KUKA KRL program: MyProgram_216().src

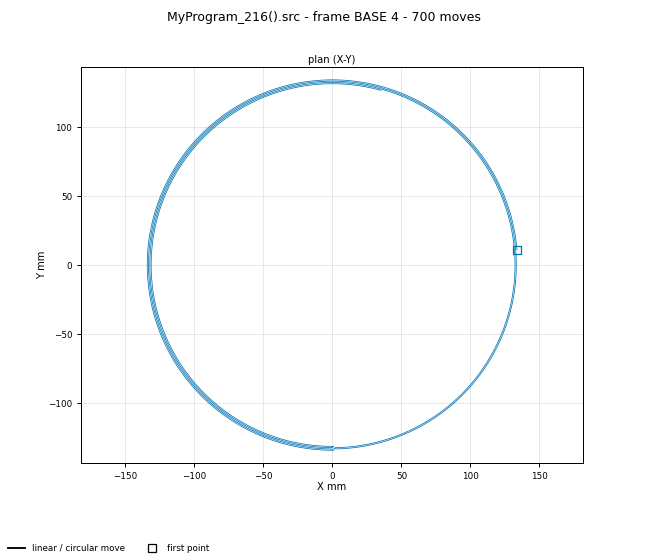
[picture p0: tool path of MyProgram_216().src in frame BASE 4, 700 of 700 moves have a stored position in this frame; points joined in program order, loops and branches not executed]
&ACCESS RVP
&REL 1
&PARAM TEMPLATE = C:\KRC\Roboter\Template\vorgabe
&PARAM EDITMASK = *
DEF MyProgram_216()
; ---- Setting reference (Base) ----
$BASE = BASE_DATA[4]

; --------------------------
; ---- Setting tool (TCP) ----
$TOOL = TOOL_DATA[3]
; --------------------------

$VEL.CP = VEL_APROX_PRINT
Startdeposition()
$VEL.CP = VEL_PRINT
LIN {X 133.7313,Y 11.0873,Z 152,A 1.5127,B 24.9579,C -1.4999,E1 25.1592,E2 444.9468} C_DIS
LIN {X 133.4155,Y 14.396,Z 152,A 2.9886,B 24.9574,C -1.5078,E1 25.1587,E2 443.4612} C_DIS
LIN {X 132.9448,Y 18.2524,Z 152,A 4.7216,B 24.9569,C -1.5174,E1 25.1581,E2 441.7159} C_DIS
LIN {X 132.4358,Y 21.6308,Z 152,A 6.0104,B 24.9571,C -1.5126,E1 25.1576,E2 440.446} C_DIS
LIN {X 131.8421,Y 24.9924,Z 152,A 7.5184,B 24.9567,C -1.5201,E1 25.1568,E2 438.9291} C_DIS
LIN {X 131.1946,Y 28.1941,Z 152,A 8.8428,B 24.9567,C -1.5206,E1 25.156,E2 437.6112} C_DIS
LIN {X 130.4813,Y 31.3296,Z 152,A 10.2545,B 24.9563,C -1.5272,E1 25.1551,E2 436.1923} C_DIS
LIN {X 129.7343,Y 34.2927,Z 152,A 11.61,B 24.9559,C -1.5341,E1 25.1542,E2 434.8282} C_DIS
LIN {X 128.7032,Y 37.9795,Z 152,A 13.1947,B 24.9558,C -1.5364,E1 25.153,E2 433.2471} C_DIS
LIN {X 127.4835,Y 41.8939,Z 152,A 14.9747,B 24.9554,C -1.5435,E1 25.1514,E2 431.4606} C_DIS
LIN {X 126.3534,Y 45.1861,Z 152,A 16.3661,B 24.9554,C -1.5427,E1 25.1502,E2 430.0789} C_DIS
LIN {X 125.2613,Y 48.1324,Z 152,A 17.8112,B 24.9548,C -1.5525,E1 25.1487,E2 428.6186} C_DIS
LIN {X 123.987,Y 51.3249,Z 152,A 19.2654,B 24.9546,C -1.5562,E1 25.1472,E2 427.1639} C_DIS
LIN {X 122.6392,Y 54.4665,Z 152,A 20.5859,B 24.9548,C -1.5527,E1 25.1457,E2 425.8588} C_DIS
LIN {X 121.2451,Y 57.5031,Z 152,A 22.076,B 24.9544,C -1.5604,E1 25.1439,E2 424.3586} C_DIS
LIN {X 119.8144,Y 60.4284,Z 152,A 23.4608,B 24.9542,C -1.5641,E1 25.1422,E2 422.9724} C_DIS
LIN {X 118.1627,Y 63.5998,Z 152,A 24.9583,B 24.954,C -1.5667,E1 25.1403,E2 421.4766} C_DIS
LIN {X 116.2257,Y 67.0745,Z 152,A 26.7209,B 24.9535,C -1.575,E1 25.1378,E2 419.7036} C_DIS
LIN {X 114.0335,Y 70.7371,Z 152,A 28.4898,B 24.9535,C -1.577,E1 25.1352,E2 417.9391} C_DIS
LIN {X 111.8163,Y 74.193,Z 152,A 30.2878,B 24.953,C -1.5841,E1 25.1325,E2 416.1331} C_DIS
LIN {X 109.4013,Y 77.7103,Z 152,A 32.1022,B 24.9527,C -1.5885,E1 25.1296,E2 414.3175} C_DIS
LIN {X 106.8036,Y 81.2433,Z 152,A 33.9859,B 24.9524,C -1.5938,E1 25.1264,E2 412.4301} C_DIS
LIN {X 104.2349,Y 84.5136,Z 152,A 35.6507,B 24.9525,C -1.592,E1 25.1235,E2 410.7773} C_DIS
LIN {X 101.537,Y 87.7362,Z 152,A 37.4625,B 24.9522,C -1.5973,E1 25.1203,E2 408.9614} C_DIS
LIN {X 98.7559,Y 90.855,Z 152,A 39.2295,B 24.952,C -1.6005,E1 25.117,E2 407.1947} C_DIS
LIN {X 95.9879,Y 93.775,Z 152,A 40.9822,B 24.9517,C -1.6063,E1 25.1135,E2 405.4359} C_DIS
LIN {X 93.1738,Y 96.5714,Z 152,A 42.6108,B 24.9517,C -1.6063,E1 25.1103,E2 403.8139} C_DIS
LIN {X 90.3468,Y 99.2213,Z 152,A 44.2646,B 24.9514,C -1.6098,E1 25.1069,E2 402.1588} C_DIS
LIN {X 87.5654,Y 101.6841,Z 152,A 45.9253,B 24.951,C -1.6171,E1 25.1034,E2 400.4874} C_DIS
LIN {X 83.9511,Y 104.6886,Z 152,A 47.8636,B 24.951,C -1.6171,E1 25.0992,E2 398.5561} C_DIS
LIN {X 80.9004,Y 107.063,Z 152,A 49.53,B 24.9508,C -1.6211,E1 25.0955,E2 396.8865} C_DIS
LIN {X 77.4008,Y 109.6196,Z 152,A 51.379,B 24.9506,C -1.6243,E1 25.0913,E2 395.0364} C_DIS
LIN {X 73.8298,Y 112.0559,Z 152,A 53.2038,B 24.9504,C -1.6263,E1 25.0871,E2 393.2132} C_DIS
LIN {X 70.4565,Y 114.2075,Z 152,A 54.9256,B 24.9502,C -1.6297,E1 25.083,E2 391.4888} C_DIS
LIN {X 67.0207,Y 116.2568,Z 152,A 56.6299,B 24.9501,C -1.6321,E1 25.0789,E2 389.7841} C_DIS
LIN {X 63.2307,Y 118.361,Z 152,A 58.4829,B 24.9499,C -1.6348,E1 25.0744,E2 387.93} C_DIS
LIN {X 59.7834,Y 120.1374,Z 152,A 60.1274,B 24.9499,C -1.6364,E1 25.0703,E2 386.2863} C_DIS
LIN {X 56.5816,Y 121.6776,Z 152,A 61.5102,B 24.9502,C -1.631,E1 25.0668,E2 384.9197} C_DIS
LIN {X 53.2944,Y 123.1525,Z 152,A 63.0006,B 24.9502,C -1.6302,E1 25.063,E2 383.4348} C_DIS
LIN {X 50.1244,Y 124.4765,Z 152,A 64.5712,B 24.9498,C -1.6373,E1 25.0589,E2 381.851} C_DIS
LIN {X 46.3326,Y 125.9395,Z 152,A 66.2773,B 24.9498,C -1.6374,E1 25.0545,E2 380.1483} C_DIS
LIN {X 43.1022,Y 127.0811,Z 152,A 67.8485,B 24.9493,C -1.6445,E1 25.0503,E2 378.5634} C_DIS
LIN {X 39.4563,Y 128.258,Z 152,A 69.3935,B 24.9495,C -1.6411,E1 25.0462,E2 377.0294} C_DIS
LIN {X 35.9558,Y 129.283,Z 152,A 70.9825,B 24.9494,C -1.6439,E1 25.0419,E2 375.4365} C_DIS
LIN {X 31.7004,Y 130.3919,Z 152,A 72.7739,B 24.9496,C -1.6404,E1 25.0371,E2 373.6559} C_DIS
LIN {X 28.3792,Y 131.1546,Z 152,A 74.2645,B 24.9494,C -1.6431,E1 25.033,E2 372.161} C_DIS
LIN {X 24.8262,Y 131.8739,Z 152,A 75.9447,B 24.9489,C -1.6508,E1 25.0284,E2 370.4646} C_DIS
LIN {X 20.913,Y 132.5508,Z 152,A 77.5552,B 24.9492,C -1.6468,E1 25.024,E2 368.865} C_DIS
LIN {X 17.2525,Y 133.0764,Z 152,A 79.1159,B 24.9492,C -1.6463,E1 25.0197,E2 367.307} C_DIS
LIN {X 12.8731,Y 133.5711,Z 152,A 80.9369,B 24.9494,C -1.6434,E1 25.0146,E2 365.4941} C_DIS
LIN {X 9.2958,Y 133.8685,Z 152,A 82.5431,B 24.9492,C -1.6473,E1 25.0101,E2 363.8794} C_DIS
LIN {X 5.4111,Y 134.081,Z 152,A 84.1584,B 24.9493,C -1.6448,E1 25.0056,E2 362.2704} C_DIS
LIN {X 1.5384,Y 134.1831,Z 152,A 85.898,B 24.949,C -1.6491,E1 25.0008,E2 360.5211} C_DIS
LIN {X -2.3618,Y 134.1694,Z 152,A 87.5071,B 24.9492,C -1.6458,E1 24.9963,E2 358.9198} C_DIS
LIN {X -6.3709,Y 134.0392,Z 152,A 89.2472,B 24.9492,C -1.6466,E1 24.9914,E2 357.1773} C_DIS
LIN {X -10.1962,Y 133.8028,Z 152,A 90.829,B 24.9494,C -1.6431,E1 24.987,E2 355.6033} C_DIS
LIN {X -14.1568,Y 133.4413,Z 152,A 92.4422,B 24.9497,C -1.6378,E1 24.9826,E2 354.0017} C_DIS
LIN {X -16.9888,Y 133.1109,Z 152,A 93.8388,B 24.9492,C -1.6464,E1 24.9787,E2 352.5839} C_DIS
LIN {X -20.9159,Y 132.5504,Z 152,A 95.4997,B 24.9494,C -1.6435,E1 24.9741,E2 350.9283} C_DIS
LIN {X -24.8462,Y 131.87,Z 152,A 97.0933,B 24.9498,C -1.6365,E1 24.9698,E2 349.3497} C_DIS
LIN {X -28.2027,Y 131.1927,Z 152,A 98.6253,B 24.9497,C -1.6389,E1 24.9655,E2 347.8102} C_DIS
LIN {X -31.5524,Y 130.4276,Z 152,A 100.1386,B 24.9497,C -1.6399,E1 24.9614,E2 346.2926} C_DIS
LIN {X -35.7751,Y 129.3336,Z 152,A 102.0205,B 24.9497,C -1.6389,E1 24.9563,E2 344.4101} C_DIS
LIN {X -39.2856,Y 128.3102,Z 152,A 103.4854,B 24.9501,C -1.6322,E1 24.9525,E2 342.9587} C_DIS
LIN {X -42.0322,Y 127.4375,Z 152,A 104.8372,B 24.9498,C -1.6369,E1 24.9488,E2 341.5932} C_DIS
LIN {X -45.8569,Y 126.1116,Z 152,A 106.5663,B 24.9499,C -1.6347,E1 24.9443,E2 339.8659} C_DIS
LIN {X -49.5966,Y 124.6892,Z 152,A 108.286,B 24.95,C -1.6329,E1 24.9398,E2 338.1469} C_DIS
LIN {X -53.1698,Y 123.2064,Z 152,A 109.8139,B 24.9506,C -1.6242,E1 24.9359,E2 336.6361} C_DIS
LIN {X -56.2408,Y 121.8352,Z 152,A 111.2411,B 24.9507,C -1.6215,E1 24.9323,E2 335.2117} C_DIS
LIN {X -59.2294,Y 120.4107,Z 152,A 112.6995,B 24.9507,C -1.6215,E1 24.9286,E2 333.7495} C_DIS
LIN {X -62.2741,Y 118.8645,Z 152,A 114.1552,B 24.9509,C -1.6189,E1 24.925,E2 332.2961} C_DIS
LIN {X -65.655,Y 117.0333,Z 152,A 115.9269,B 24.9507,C -1.6226,E1 24.9207,E2 330.5107} C_DIS
LIN {X -69.6111,Y 114.7244,Z 152,A 117.8168,B 24.9511,C -1.6156,E1 24.9162,E2 328.6315} C_DIS
LIN {X -72.8488,Y 112.6964,Z 152,A 119.5085,B 24.9511,C -1.6155,E1 24.9122,E2 326.9348} C_DIS
LIN {X -76.4014,Y 110.3189,Z 152,A 121.2229,B 24.9517,C -1.6062,E1 24.9082,E2 325.2366} C_DIS
LIN {X -80.5,Y 107.3651,Z 152,A 123.7555,B 24.9508,C -1.6205,E1 24.9024,E2 322.661} C_DIS
LIN {X -83.2101,Y 105.2786,Z 152,A 124.9589,B 24.9518,C -1.6044,E1 24.8999,E2 321.4916} C_DIS
LIN {X -86.56,Y 102.542,Z 152,A 126.6153,B 24.9526,C -1.5907,E1 24.8964,E2 319.8614} C_DIS
LIN {X -89.6519,Y 99.8494,Z 152,A 128.5412,B 24.9523,C -1.5954,E1 24.8923,E2 317.9169} C_DIS
LIN {X -92.4999,Y 97.2173,Z 152,A 130.213,B 24.9525,C -1.5922,E1 24.8889,E2 316.2458} C_DIS
LIN {X -95.3781,Y 94.3951,Z 152,A 131.9585,B 24.9527,C -1.5891,E1 24.8854,E2 314.5001} C_DIS
LIN {X -99.147,Y 90.4287,Z 152,A 134.3393,B 24.9529,C -1.5854,E1 24.8809,E2 312.1178} C_DIS
LIN {X -101.8173,Y 87.4107,Z 152,A 136.0686,B 24.9531,C -1.5813,E1 24.8777,E2 310.3904} C_DIS
LIN {X -104.5409,Y 84.1343,Z 152,A 137.8461,B 24.9536,C -1.5744,E1 24.8746,E2 308.6213} C_DIS
LIN {X -107.0195,Y 80.958,Z 152,A 139.593,B 24.9538,C -1.571,E1 24.8716,E2 306.874} C_DIS
LIN {X -109.3032,Y 77.8474,Z 152,A 141.2807,B 24.9539,C -1.5683,E1 24.8689,E2 305.1844} C_DIS
LIN {X -111.7611,Y 74.2757,Z 152,A 143.0987,B 24.9543,C -1.5614,E1 24.866,E2 303.3739} C_DIS
LIN {X -113.9277,Y 70.9071,Z 152,A 144.8218,B 24.9546,C -1.5571,E1 24.8635,E2 301.6523} C_DIS
LIN {X -115.9039,Y 67.6298,Z 152,A 146.5135,B 24.9546,C -1.5551,E1 24.861,E2 299.9566} C_DIS
LIN {X -117.7597,Y 64.3429,Z 152,A 148.0857,B 24.9551,C -1.5484,E1 24.8589,E2 298.3922} C_DIS
LIN {X -119.5065,Y 61.0332,Z 152,A 149.6708,B 24.9554,C -1.5429,E1 24.8569,E2 296.8116} C_DIS
LIN {X -121.0233,Y 57.9674,Z 152,A 151.1342,B 24.9556,C -1.5386,E1 24.8551,E2 295.3505} C_DIS
LIN {X -122.4213,Y 54.9536,Z 152,A 152.4985,B 24.9561,C -1.5316,E1 24.8535,E2 293.9956} C_DIS
LIN {X -123.7101,Y 51.9879,Z 152,A 153.9859,B 24.956,C -1.5325,E1 24.8519,E2 292.4977} C_DIS
LIN {X -124.9732,Y 48.8736,Z 152,A 155.4287,B 24.9562,C -1.5284,E1 24.8504,E2 291.0567} C_DIS
LIN {X -126.2429,Y 45.4928,Z 152,A 156.9066,B 24.9567,C -1.5203,E1 24.849,E2 289.5896} C_DIS
LIN {X -127.1836,Y 42.7946,Z 152,A 158.2602,B 24.9565,C -1.523,E1 24.8478,E2 288.222} C_DIS
LIN {X -128.3048,Y 39.3032,Z 152,A 159.6429,B 24.9573,C -1.509,E1 24.8466,E2 286.8647} C_DIS
LIN {X -129.2501,Y 36.0735,Z 152,A 161.2232,B 24.9573,C -1.5114,E1 24.8454,E2 285.2695} C_DIS
LIN {X -130.2973,Y 32.0928,Z 152,A 162.9399,B 24.9576,C -1.5036,E1 24.8442,E2 283.5613} C_DIS
LIN {X -131.1463,Y 28.4176,Z 152,A 164.5492,B 24.9579,C -1.4983,E1 24.8432,E2 281.9552} C_DIS
LIN {X -131.7346,Y 25.5545,Z 152,A 165.8929,B 24.9579,C -1.4989,E1 24.8425,E2 280.6022} C_DIS
LIN {X -132.3897,Y 21.9072,Z 152,A 167.4388,B 24.9583,C -1.4919,E1 24.8418,E2 279.0637} C_DIS
LIN {X -132.9993,Y 17.8409,Z 152,A 169.204,B 24.9586,C -1.4866,E1 24.8411,E2 277.3007} C_DIS
LIN {X -133.4252,Y 14.306,Z 152,A 170.7541,B 24.9588,C -1.483,E1 24.8406,E2 275.7498} C_DIS
LIN {X -133.79,Y 10.371,Z 152,A 172.5007,B 24.9589,C -1.4804,E1 24.8402,E2 273.9991} C_DIS
LIN {X -134.0268,Y 6.618,Z 152,A 174.0782,B 24.9593,C -1.4737,E1 24.8399,E2 272.428} C_DIS
LIN {X -134.1689,Y 2.3895,Z 152,A 175.8019,B 24.9599,C -1.4636,E1 24.8399,E2 270.7179} C_DIS
LIN {X -134.1918,Y -0.3012,Z 152,A 177.13,B 24.9596,C -1.4686,E1 24.8398,E2 269.3699} C_DIS
LIN {X -134.1223,Y -4.3022,Z 152,A 178.8913,B 24.9598,C -1.4656,E1 24.8399,E2 267.6052} C_DIS
LIN {X -133.9167,Y -8.5657,Z 152,A -179.4068,B 24.9604,C -1.4537,E1 24.8402,E2 265.9215} C_DIS
LIN {X -133.5825,Y -12.7544,Z 152,A -177.6549,B 24.9608,C -1.4457,E1 24.8406,E2 264.178} C_DIS
LIN {X -133.2718,Y -15.6723,Z 152,A -176.3213,B 24.9608,C -1.4456,E1 24.841,E2 262.8367} C_DIS
LIN {X -132.8013,Y -19.2565,Z 152,A -174.7809,B 24.9611,C -1.4404,E1 24.8416,E2 261.2994} C_DIS
LIN {X -132.3608,Y -22.0803,Z 152,A -172.8087,B 24.9593,C -1.4738,E1 24.8426,E2 259.2359} C_DIS
LIN {X -131.2989,Y -27.7109,Z 152,A -171.0218,B 24.9615,C -1.4331,E1 24.8435,E2 257.5354} C_DIS
LIN {X -130.5269,Y -31.1405,Z 152,A -169.5404,B 24.9618,C -1.4274,E1 24.8445,E2 256.059} C_DIS
LIN {X -129.5266,Y -35.0715,Z 152,A -167.7832,B 24.9621,C -1.4232,E1 24.8457,E2 254.3015} C_DIS
LIN {X -128.4165,Y -38.9384,Z 152,A -166.0652,B 24.9623,C -1.4179,E1 24.8471,E2 252.5862} C_DIS
LIN {X -127.3727,Y -42.2266,Z 152,A -164.6402,B 24.9627,C -1.411,E1 24.8483,E2 251.1695} C_DIS
LIN {X -126.2249,Y -45.5425,Z 152,A -163.2148,B 24.9631,C -1.4029,E1 24.8496,E2 249.7555} C_DIS
LIN {X -125.2451,Y -48.1742,Z 152,A -161.8357,B 24.9629,C -1.4082,E1 24.851,E2 248.356} C_DIS
LIN {X -124.0022,Y -51.2886,Z 152,A -160.3981,B 24.9631,C -1.4042,E1 24.8525,E2 246.9199} C_DIS
LIN {X -122.6867,Y -54.3602,Z 152,A -158.9604,B 24.9633,C -1.4005,E1 24.8541,E2 245.483} C_DIS
LIN {X -121.3107,Y -57.3657,Z 152,A -157.5589,B 24.9635,C -1.3959,E1 24.8558,E2 244.0848} C_DIS
LIN {X -119.7947,Y -60.467,Z 152,A -156.0476,B 24.9636,C -1.3936,E1 24.8577,E2 242.5709} C_DIS
LIN {X -118.0171,Y -63.8709,Z 152,A -154.4079,B 24.9639,C -1.389,E1 24.8598,E2 240.9336} C_DIS
LIN {X -116.0917,Y -67.3059,Z 152,A -152.7725,B 24.9642,C -1.382,E1 24.8621,E2 239.3061} C_DIS
LIN {X -114.075,Y -70.6706,Z 152,A -150.994,B 24.9642,C -1.3827,E1 24.8647,E2 237.5169} C_DIS
LIN {X -111.5754,Y -74.5539,Z 152,A -149.1002,B 24.9647,C -1.3735,E1 24.8676,E2 235.6354} C_DIS
LIN {X -109.2915,Y -77.8638,Z 152,A -147.473,B 24.9651,C -1.3646,E1 24.8701,E2 234.0215} C_DIS
LIN {X -106.7329,Y -81.3357,Z 152,A -145.444,B 24.9649,C -1.3694,E1 24.8736,E2 231.9712} C_DIS
LIN {X -103.909,Y -84.9133,Z 152,A -143.5748,B 24.9653,C -1.3608,E1 24.8768,E2 230.1139} C_DIS
LIN {X -101.4481,Y -87.8394,Z 152,A -141.8793,B 24.9653,C -1.3601,E1 24.8799,E2 228.4123} C_DIS
LIN {X -98.7806,Y -90.8281,Z 152,A -140.2022,B 24.9656,C -1.3545,E1 24.883,E2 226.7411} C_DIS
LIN {X -96.4069,Y -93.3438,Z 152,A -138.6921,B 24.9657,C -1.3529,E1 24.886,E2 225.2283} C_DIS
LIN {X -93.286,Y -96.4628,Z 152,A -136.7804,B 24.9659,C -1.3502,E1 24.8898,E2 223.3148} C_DIS
LIN {X -90.1471,Y -99.4025,Z 152,A -134.9589,B 24.9661,C -1.3456,E1 24.8935,E2 221.4969} C_DIS
LIN {X -87.0495,Y -102.1263,Z 152,A -133.2129,B 24.9663,C -1.3414,E1 24.8972,E2 219.7542} C_DIS
LIN {X -83.9461,Y -104.6926,Z 152,A -131.4446,B 24.9663,C -1.3406,E1 24.901,E2 217.9812} C_DIS
LIN {X -78.6575,Y -108.7214,Z 152,A -128.6331,B 24.9667,C -1.334,E1 24.9073,E2 215.1751} C_DIS
LIN {X -75.474,Y -110.9555,Z 152,A -126.8798,B 24.9666,C -1.336,E1 24.9114,E2 213.4112} C_DIS
LIN {X -71.8364,Y -113.3443,Z 152,A -125.0645,B 24.9668,C -1.3308,E1 24.9156,E2 211.6024} C_DIS
LIN {X -68.2007,Y -115.5686,Z 152,A -123.2173,B 24.9668,C -1.3295,E1 24.92,E2 209.7527} C_DIS
LIN {X -64.4441,Y -117.7045,Z 152,A -121.4191,B 24.9671,C -1.3245,E1 24.9244,E2 207.9612} C_DIS
LIN {X -61.1288,Y -119.4578,Z 152,A -119.9025,B 24.9675,C -1.318,E1 24.9281,E2 206.4558} C_DIS
LIN {X -57.8791,Y -121.0655,Z 152,A -118.3995,B 24.9677,C -1.3137,E1 24.9319,E2 204.959} C_DIS
LIN {X -55.2881,Y -122.2717,Z 152,A -117.0006,B 24.9673,C -1.3216,E1 24.9355,E2 203.5381} C_DIS
LIN {X -52.1484,Y -123.6431,Z 152,A -115.5975,B 24.9675,C -1.3169,E1 24.9391,E2 202.1429} C_DIS
LIN {X -48.7188,Y -125.0334,Z 152,A -114.1694,B 24.968,C -1.3074,E1 24.9427,E2 200.7342} C_DIS
LIN {X -45.6153,Y -126.1987,Z 152,A -112.6719,B 24.9678,C -1.3103,E1 24.9467,E2 199.2267} C_DIS
LIN {X -42.3577,Y -127.3291,Z 152,A -111.1317,B 24.9678,C -1.3126,E1 24.9508,E2 197.6781} C_DIS
LIN {X -38.4982,Y -128.5512,Z 152,A -109.2547,B 24.9674,C -1.3191,E1 24.9558,E2 195.7825} C_DIS
LIN {X -34.526,Y -129.6721,Z 152,A -107.6238,B 24.9678,C -1.311,E1 24.9602,E2 194.1681} C_DIS
LIN {X -30.7102,Y -130.6306,Z 152,A -105.8521,B 24.9676,C -1.3149,E1 24.965,E2 192.3848} C_DIS
LIN {X -26.8072,Y -131.4849,Z 152,A -104.2939,B 24.968,C -1.3064,E1 24.9692,E2 190.8449} C_DIS
LIN {X -23.8231,Y -132.0584,Z 152,A -103.0446,B 24.9682,C -1.3033,E1 24.9726,E2 189.6016} C_DIS
LIN {X -20.7101,Y -132.5822,Z 152,A -101.6459,B 24.9681,C -1.3056,E1 24.9765,E2 188.1961} C_DIS
LIN {X -17.6843,Y -133.0198,Z 152,A -100.2691,B 24.9679,C -1.3091,E1 24.9803,E2 186.81} C_DIS
LIN {X -13.8573,Y -133.4735,Z 152,A -98.5314,B 24.9677,C -1.3138,E1 24.9852,E2 185.0601} C_DIS
LIN {X -9.8697,Y -133.8266,Z 152,A -96.9829,B 24.9681,C -1.3052,E1 24.9895,E2 183.5314} C_DIS
LIN {X -6.8034,Y -134.0175,Z 152,A -95.5784,B 24.9678,C -1.3102,E1 24.9934,E2 182.1146} C_DIS
LIN {X -2.6797,Y -134.1641,Z 152,A -93.7877,B 24.9678,C -1.312,E1 24.9984,E2 180.3194} C_DIS
LIN {X 0.9471,Y -134.1856,Z 152,A -92.9028,B 24.9695,C -1.277,E1 25.0007,E2 179.5173} C_DIS
Enddeposition()
LIN {X 0.9471,Y -134.1856,Z 152,A -92.9028,B 24.9695,C -1.277,E1 25.0007,E2 179.5173} C_DIS
Startdeposition()
$VEL.CP = VEL_PRINT
LIN {X -0.5929,Y -133.247,Z 152,A -93.69,B 24.8761,C -1.2672,E1 24.9047,E2 180.3158} C_DIS
LIN {X -4.8796,Y -133.1592,Z 152,A -95.4999,B 24.876,C -1.2687,E1 24.8997,E2 182.1224} C_DIS
LIN {X -8.6167,Y -132.97,Z 152,A -97.2057,B 24.8762,C -1.2636,E1 24.8949,E2 183.8408} C_DIS
LIN {X -12.6109,Y -132.6501,Z 152,A -98.8357,B 24.876,C -1.2685,E1 24.8904,E2 185.4599} C_DIS
LIN {X -16.5782,Y -132.2149,Z 152,A -100.6527,B 24.8762,C -1.2635,E1 24.8853,E2 187.2899} C_DIS
LIN {X -20.1629,Y -131.7139,Z 152,A -102.1207,B 24.876,C -1.2685,E1 24.8813,E2 188.7473} C_DIS
LIN {X -23.7027,Y -131.1231,Z 152,A -103.6682,B 24.876,C -1.2688,E1 24.877,E2 190.2956} C_DIS
LIN {X -27.9153,Y -130.2912,Z 152,A -105.4125,B 24.8757,C -1.2748,E1 24.8723,E2 192.0276} C_DIS
LIN {X -31.017,Y -129.5878,Z 152,A -106.8525,B 24.8758,C -1.2718,E1 24.8683,E2 193.4766} C_DIS
LIN {X -34.2778,Y -128.7635,Z 152,A -108.2404,B 24.8757,C -1.2757,E1 24.8646,E2 194.8573} C_DIS
LIN {X -37.8213,Y -127.7681,Z 152,A -109.7774,B 24.8755,C -1.2791,E1 24.8605,E2 196.3888} C_DIS
LIN {X -45.252,Y -125.3285,Z 152,A -113.3268,B 24.8758,C -1.2724,E1 24.851,E2 199.9609} C_DIS
LIN {X -49.5093,Y -123.7089,Z 152,A -115.2469,B 24.8756,C -1.2762,E1 24.846,E2 201.8759} C_DIS
LIN {X -52.7769,Y -122.3502,Z 152,A -116.6598,B 24.8753,C -1.2834,E1 24.8424,E2 203.2751} C_DIS
LIN {X -55.7134,Y -121.0414,Z 152,A -118.0747,B 24.8753,C -1.2834,E1 24.8388,E2 204.6935} C_DIS
LIN {X -58.7098,Y -119.6168,Z 152,A -119.5751,B 24.8753,C -1.2814,E1 24.835,E2 206.2025} C_DIS
LIN {X -62.5075,Y -117.6782,Z 152,A -121.6268,B 24.8758,C -1.2728,E1 24.8299,E2 208.2802} C_DIS
LIN {X -66.957,Y -115.2054,Z 152,A -123.6951,B 24.8754,C -1.282,E1 24.8249,E2 210.3328} C_DIS
LIN {X -70.7642,Y -112.9074,Z 152,A -125.6311,B 24.8753,C -1.2837,E1 24.8203,E2 212.2708} C_DIS
LIN {X -74.294,Y -110.6165,Z 152,A -127.4512,B 24.8752,C -1.2861,E1 24.816,E2 214.091} C_DIS
LIN {X -78.0168,Y -108.0226,Z 152,A -129.3098,B 24.8748,C -1.2941,E1 24.8118,E2 215.937} C_DIS
LIN {X -81.4917,Y -105.4258,Z 152,A -131.248,B 24.8748,C -1.2939,E1 24.8075,E2 217.8829} C_DIS
LIN {X -84.9957,Y -102.6216,Z 152,A -133.154,B 24.8745,C -1.2987,E1 24.8034,E2 219.7845} C_DIS
LIN {X -87.7193,Y -100.3036,Z 152,A -134.7415,B 24.8745,C -1.2993,E1 24.8,E2 221.3767} C_DIS
LIN {X -90.456,Y -97.8433,Z 152,A -137.2798,B 24.8766,C -1.2559,E1 24.7947,E2 224.0291} C_DIS
LIN {X -95.5831,Y -92.8406,Z 152,A -139.4357,B 24.8741,C -1.3076,E1 24.7906,E2 226.0707} C_DIS
LIN {X -98.7018,Y -89.5177,Z 152,A -141.3815,B 24.8739,C -1.3128,E1 24.7869,E2 228.0129} C_DIS
LIN {X -101.3494,Y -86.5092,Z 152,A -143.1336,B 24.8737,C -1.3154,E1 24.7837,E2 229.7667} C_DIS
LIN {X -104.4545,Y -82.7335,Z 152,A -145.8647,B 24.875,C -1.2899,E1 24.7788,E2 232.5714} C_DIS
LIN {X -107.7707,Y -78.3644,Z 152,A -147.6157,B 24.8732,C -1.3253,E1 24.7761,E2 234.2464} C_DIS
LIN {X -110.4537,Y -74.5352,Z 152,A -149.5668,B 24.8728,C -1.3334,E1 24.773,E2 236.1878} C_DIS
LIN {X -112.7814,Y -70.9637,Z 152,A -151.4618,B 24.8728,C -1.3353,E1 24.7701,E2 238.0879} C_DIS
LIN {X -115.0943,Y -67.1485,Z 152,A -153.4018,B 24.8725,C -1.3395,E1 24.7673,E2 240.0281} C_DIS
LIN {X -117.1845,Y -63.4305,Z 152,A -155.283,B 24.8724,C -1.3423,E1 24.7648,E2 241.9124} C_DIS
LIN {X -119.2529,Y -59.4475,Z 152,A -157.1605,B 24.872,C -1.3503,E1 24.7624,E2 243.7808} C_DIS
LIN {X -120.884,Y -56.0538,Z 152,A -158.7067,B 24.8715,C -1.3586,E1 24.7606,E2 245.3158} C_DIS
LIN {X -122.2811,Y -52.9367,Z 152,A -160.1631,B 24.8713,C -1.3635,E1 24.759,E2 246.7685} C_DIS
LIN {X -123.4892,Y -50.0544,Z 152,A -161.5135,B 24.8711,C -1.3671,E1 24.7575,E2 248.1177} C_DIS
LIN {X -124.6583,Y -47.0681,Z 152,A -162.9823,B 24.8711,C -1.3669,E1 24.756,E2 249.5952} C_DIS
LIN {X -125.7882,Y -43.9593,Z 152,A -164.3822,B 24.8708,C -1.3723,E1 24.7547,E2 250.9903} C_DIS
LIN {X -126.8893,Y -40.6707,Z 152,A -165.8542,B 24.8706,C -1.3778,E1 24.7535,E2 252.4575} C_DIS
LIN {X -127.8411,Y -37.5723,Z 152,A -167.2897,B 24.8704,C -1.3801,E1 24.7523,E2 253.8959} C_DIS
LIN {X -128.7838,Y -34.2019,Z 152,A -168.797,B 24.8702,C -1.3847,E1 24.7512,E2 255.401} C_DIS
LIN {X -129.7494,Y -30.3409,Z 152,A -170.6146,B 24.8702,C -1.385,E1 24.75,E2 257.2285} C_DIS
LIN {X -130.5583,Y -26.6376,Z 152,A -172.1168,B 24.8696,C -1.3964,E1 24.7491,E2 258.7125} C_DIS
LIN {X -131.1897,Y -23.3307,Z 152,A -173.7196,B 24.8697,C -1.3936,E1 24.7483,E2 260.3316} C_DIS
LIN {X -131.8769,Y -19.0677,Z 152,A -175.4614,B 24.8691,C -1.4051,E1 24.7476,E2 262.0564} C_DIS
LIN {X -132.7751,Y -11.2186,Z 152,A -178.907,B 24.8687,C -1.4138,E1 24.7466,E2 265.5018} C_DIS
LIN {X -133.0574,Y -7.1421,Z 152,A 179.2854,B 24.8685,C -1.4171,E1 24.7462,E2 267.3123} C_DIS
LIN {X -133.2014,Y -3.5382,Z 152,A 177.7117,B 24.8683,C -1.4211,E1 24.7461,E2 268.8859} C_DIS
LIN {X -133.2493,Y 0.4133,Z 152,A 175.9894,B 24.868,C -1.4256,E1 24.7461,E2 270.608} C_DIS
LIN {X -133.1759,Y 4.4518,Z 152,A 174.1957,B 24.8679,C -1.4286,E1 24.7461,E2 272.4053} C_DIS
LIN {X -132.995,Y 8.2106,Z 152,A 172.6437,B 24.8674,C -1.4372,E1 24.7464,E2 273.9462} C_DIS
LIN {X -132.668,Y 12.4241,Z 152,A 170.7948,B 24.8672,C -1.4417,E1 24.7469,E2 275.7956} C_DIS
LIN {X -132.2426,Y 16.3483,Z 152,A 169.0088,B 24.8671,C -1.443,E1 24.7475,E2 277.5891} C_DIS
LIN {X -131.6821,Y 20.3682,Z 152,A 167.3798,B 24.8665,C -1.4543,E1 24.7481,E2 279.2007} C_DIS
LIN {X -131.1882,Y 23.339,Z 152,A 166.1859,B 24.866,C -1.4634,E1 24.7487,E2 280.38} C_DIS
LIN {X -130.0151,Y 29.1779,Z 152,A 163.454,B 24.866,C -1.4636,E1 24.7502,E2 283.1277} C_DIS
LIN {X -129.1811,Y 32.669,Z 152,A 161.9442,B 24.8656,C -1.4702,E1 24.7512,E2 284.6305} C_DIS
LIN {X -128.293,Y 35.9989,Z 152,A 160.473,B 24.8653,C -1.4755,E1 24.7523,E2 286.0975} C_DIS
LIN {X -127.3218,Y 39.297,Z 152,A 158.947,B 24.8652,C -1.478,E1 24.7535,E2 287.6265} C_DIS
LIN {X -126.0023,Y 43.3417,Z 152,A 157.0976,B 24.8649,C -1.4829,E1 24.7552,E2 289.4748} C_DIS
LIN {X -124.8348,Y 46.5968,Z 152,A 155.6073,B 24.8646,C -1.4875,E1 24.7566,E2 290.9627} C_DIS
LIN {X -123.5338,Y 49.9438,Z 152,A 154.1021,B 24.8643,C -1.4942,E1 24.7581,E2 292.4603} C_DIS
LIN {X -121.8994,Y 53.8137,Z 152,A 152.1817,B 24.8643,C -1.4943,E1 24.7603,E2 294.3911} C_DIS
LIN {X -120.2957,Y 57.3055,Z 152,A 150.4447,B 24.8642,C -1.4954,E1 24.7623,E2 296.135} C_DIS
LIN {X -116.8179,Y 64.1028,Z 152,A 147.1943,B 24.8636,C -1.5068,E1 24.7665,E2 299.3755} C_DIS
LIN {X -114.6781,Y 67.8571,Z 152,A 145.3163,B 24.8633,C -1.5113,E1 24.7691,E2 301.2524} C_DIS
LIN {X -112.4249,Y 71.528,Z 152,A 143.4234,B 24.8631,C -1.5147,E1 24.7719,E2 303.1468} C_DIS
LIN {X -109.9657,Y 75.2531,Z 152,A 141.5424,B 24.8627,C -1.5221,E1 24.7749,E2 305.0197} C_DIS
LIN {X -107.522,Y 78.7053,Z 152,A 139.6789,B 24.8625,C -1.525,E1 24.7779,E2 306.8853} C_DIS
LIN {X -104.7396,Y 82.3717,Z 152,A 137.7181,B 24.8621,C -1.5313,E1 24.7812,E2 308.8405} C_DIS
LIN {X -101.8876,Y 85.8747,Z 152,A 135.7401,B 24.8619,C -1.5347,E1 24.7848,E2 310.8194} C_DIS
LIN {X -98.9414,Y 89.2537,Z 152,A 133.8092,B 24.8617,C -1.5396,E1 24.7883,E2 312.7474} C_DIS
LIN {X -95.5752,Y 92.8487,Z 152,A 131.6832,B 24.8614,C -1.5446,E1 24.7924,E2 314.8708} C_DIS
LIN {X -92.3821,Y 96.027,Z 152,A 129.6897,B 24.8613,C -1.5466,E1 24.7964,E2 316.8679} C_DIS
LIN {X -87.2876,Y 100.6803,Z 152,A 126.7176,B 24.8609,C -1.5533,E1 24.8026,E2 319.8358} C_DIS
LIN {X -83.9393,Y 103.4881,Z 152,A 124.8282,B 24.8607,C -1.557,E1 24.8066,E2 321.7236} C_DIS
LIN {X -80.3346,Y 106.31,Z 152,A 122.9566,B 24.8601,C -1.566,E1 24.8108,E2 323.5806} C_DIS
LIN {X -76.8949,Y 108.8239,Z 152,A 121.0494,B 24.8601,C -1.5662,E1 24.8151,E2 325.4941} C_DIS
LIN {X -73.148,Y 111.3771,Z 152,A 119.1205,B 24.8598,C -1.5711,E1 24.8196,E2 327.4177} C_DIS
LIN {X -69.3847,Y 113.7601,Z 152,A 117.1567,B 24.8598,C -1.5724,E1 24.8242,E2 329.3847} C_DIS
LIN {X -65.6509,Y 115.9552,Z 152,A 115.2565,B 24.8597,C -1.5739,E1 24.8288,E2 331.2868} C_DIS
LIN {X -61.9434,Y 117.9744,Z 152,A 113.5346,B 24.8592,C -1.5817,E1 24.833,E2 332.9951} C_DIS
LIN {X -58.2975,Y 119.8202,Z 152,A 111.693,B 24.8592,C -1.5804,E1 24.8376,E2 334.8446} C_DIS
LIN {X -54.6438,Y 121.5281,Z 152,A 110.1267,B 24.8586,C -1.5914,E1 24.8416,E2 336.3886} C_DIS
LIN {X -51.5725,Y 122.8629,Z 152,A 108.5849,B 24.8588,C -1.5885,E1 24.8456,E2 337.9409} C_DIS
LIN {X -48.3257,Y 124.1757,Z 152,A 107.0871,B 24.8586,C -1.591,E1 24.8494,E2 339.4361} C_DIS
LIN {X -44.6946,Y 125.5295,Z 152,A 105.3085,B 24.8588,C -1.5876,E1 24.8541,E2 341.2264} C_DIS
LIN {X -40.6558,Y 126.8941,Z 152,A 103.6225,B 24.8583,C -1.5971,E1 24.8585,E2 342.8927} C_DIS
LIN {X -37.3842,Y 127.8961,Z 152,A 102.2404,B 24.8579,C -1.6033,E1 24.8622,E2 344.2626} C_DIS
LIN {X -32.9119,Y 129.1195,Z 152,A 100.3698,B 24.8574,C -1.6115,E1 24.8672,E2 346.1164} C_DIS
LIN {X -29.1319,Y 130.0256,Z 152,A 98.3831,B 24.8583,C -1.5972,E1 24.8727,E2 348.1397} C_DIS
LIN {X -23.7765,Y 131.1099,Z 152,A 95.9462,B 24.8584,C -1.5948,E1 24.8794,E2 350.5851} C_DIS
LIN {X -18.9901,Y 131.888,Z 152,A 94.0081,B 24.8579,C -1.6036,E1 24.8847,E2 352.5039} C_DIS
LIN {X -15.5057,Y 132.3431,Z 152,A 92.4126,B 24.8581,C -1.6003,E1 24.8892,E2 354.1085} C_DIS
LIN {X -11.2253,Y 132.7745,Z 152,A 90.6402,B 24.8578,C -1.6051,E1 24.8941,E2 355.8702} C_DIS
LIN {X -7.258,Y 133.0516,Z 152,A 88.8774,B 24.8579,C -1.6031,E1 24.899,E2 357.6384} C_DIS
LIN {X -3.5696,Y 133.2005,Z 152,A 87.3206,B 24.8578,C -1.6052,E1 24.9033,E2 359.1906} C_DIS
LIN {X 0.5929,Y 133.247,Z 152,A 85.544,B 24.8578,C -1.6062,E1 24.9083,E2 360.9647} C_DIS
LIN {X 4.5818,Y 133.1708,Z 152,A 83.7445,B 24.858,C -1.6021,E1 24.9133,E2 362.7735} C_DIS
LIN {X 8.5349,Y 132.975,Z 152,A 82.017,B 24.858,C -1.6008,E1 24.9181,E2 364.5035} C_DIS
LIN {X 12.732,Y 132.6385,Z 152,A 80.3409,B 24.8576,C -1.6075,E1 24.9228,E2 366.1626} C_DIS
LIN {X 16.293,Y 132.2492,Z 152,A 78.6802,B 24.858,C -1.6011,E1 24.9274,E2 367.8375} C_DIS
LIN {X 20.3183,Y 131.6898,Z 152,A 77.0476,B 24.8577,C -1.6065,E1 24.9319,E2 369.4557} C_DIS
LIN {X 23.8215,Y 131.1018,Z 152,A 75.4496,B 24.858,C -1.6023,E1 24.9363,E2 371.0621} C_DIS
LIN {X 27.6773,Y 130.3426,Z 152,A 73.7773,B 24.858,C -1.6023,E1 24.9409,E2 372.732} C_DIS
LIN {X 31.7159,Y 129.4194,Z 152,A 71.8575,B 24.8584,C -1.5942,E1 24.9461,E2 374.6685} C_DIS
LIN {X 34.8303,Y 128.6162,Z 152,A 69.5653,B 24.8613,C -1.5466,E1 24.9527,E2 377.0699} C_DIS
LIN {X 41.9547,Y 126.4706,Z 152,A 67.32,B 24.8585,C -1.593,E1 24.9583,E2 379.201} C_DIS
LIN {X 46.4246,Y 124.8993,Z 152,A 65.4484,B 24.8581,C -1.5997,E1 24.9631,E2 381.0527} C_DIS
LIN {X 49.5583,Y 123.6892,Z 152,A 63.9823,B 24.8583,C -1.5971,E1 24.9669,E2 382.5218} C_DIS
LIN {X 52.6203,Y 122.4179,Z 152,A 62.5652,B 24.8583,C -1.596,E1 24.9706,E2 383.9383} C_DIS
LIN {X 55.6523,Y 121.0697,Z 152,A 61.1886,B 24.8583,C -1.5969,E1 24.9741,E2 385.3092} C_DIS
LIN {X 58.5756,Y 119.683,Z 152,A 59.7861,B 24.8584,C -1.5946,E1 24.9776,E2 386.7135} C_DIS
LIN {X 62.526,Y 117.6685,Z 152,A 57.8083,B 24.8588,C -1.5882,E1 24.9825,E2 388.7008} C_DIS
LIN {X 66.3874,Y 115.5351,Z 152,A 55.8475,B 24.8592,C -1.5821,E1 24.9873,E2 390.6703} C_DIS
LIN {X 70.2092,Y 113.2527,Z 152,A 53.9726,B 24.8592,C -1.5812,E1 24.9918,E2 392.5414} C_DIS
LIN {X 73.9187,Y 110.867,Z 152,A 52.0568,B 24.8595,C -1.5771,E1 24.9963,E2 394.4606} C_DIS
LIN {X 79.4365,Y 106.9829,Z 152,A 49.1764,B 24.8597,C -1.5731,E1 25.0028,E2 397.3403} C_DIS
LIN {X 83.0142,Y 104.231,Z 152,A 47.255,B 24.8599,C -1.5705,E1 25.007,E2 399.2608} C_DIS
LIN {X 86.5099,Y 101.3488,Z 152,A 45.3231,B 24.86,C -1.5675,E1 25.0112,E2 401.1923} C_DIS
LIN {X 89.8429,Y 98.4067,Z 152,A 43.3556,B 24.8604,C -1.5606,E1 25.0153,E2 403.1683} C_DIS
LIN {X 93.2651,Y 95.1688,Z 152,A 41.4104,B 24.8604,C -1.5606,E1 25.0192,E2 405.1054} C_DIS
LIN {X 96.4059,Y 91.9857,Z 152,A 39.4973,B 24.8607,C -1.5568,E1 25.0229,E2 407.0192} C_DIS
LIN {X 99.3389,Y 88.8103,Z 152,A 37.6719,B 24.8608,C -1.5543,E1 25.0263,E2 408.8424} C_DIS
LIN {X 102.2327,Y 85.4634,Z 152,A 35.8446,B 24.8608,C -1.5538,E1 25.0296,E2 410.6625} C_DIS
LIN {X 105.0655,Y 81.9565,Z 152,A 33.7928,B 24.8615,C -1.5429,E1 25.0332,E2 412.7305} C_DIS
LIN {X 107.6826,Y 78.4859,Z 152,A 31.9265,B 24.8617,C -1.5383,E1 25.0363,E2 414.5986} C_DIS
LIN {X 109.7114,Y 75.6237,Z 152,A 30.1271,B 24.8629,C -1.5187,E1 25.0392,E2 416.4355} C_DIS
LIN {X 111.8858,Y 72.3677,Z 152,A 28.7775,B 24.8621,C -1.5323,E1 25.0412,E2 417.7463} C_DIS
LIN {X 114.164,Y 68.7177,Z 152,A 26.9586,B 24.8623,C -1.529,E1 25.0439,E2 419.5638} C_DIS
LIN {X 116.372,Y 64.9092,Z 152,A 25.0329,B 24.8627,C -1.5219,E1 25.0466,E2 421.4961} C_DIS
LIN {X 118.5243,Y 60.8865,Z 152,A 23.173,B 24.8627,C -1.5219,E1 25.049,E2 423.3461} C_DIS
LIN {X 120.053,Y 57.8135,Z 152,A 21.5012,B 24.8635,C -1.507,E1 25.051,E2 425.0442} C_DIS
LIN {X 122.1706,Y 53.1923,Z 152,A 19.5383,B 24.8632,C -1.5128,E1 25.0532,E2 426.9828} C_DIS
LIN {X 123.5059,Y 50.0131,Z 152,A 18.0817,B 24.8634,C -1.5098,E1 25.0548,E2 428.4384} C_DIS
LIN {X 124.8402,Y 46.5824,Z 152,A 16.5073,B 24.8636,C -1.5055,E1 25.0564,E2 430.0142} C_DIS
LIN {X 126.2031,Y 42.7581,Z 152,A 14.7088,B 24.8641,C -1.4972,E1 25.058,E2 431.822} C_DIS
LIN {X 127.2962,Y 39.3806,Z 152,A 13.293,B 24.8641,C -1.4986,E1 25.0592,E2 433.2266} C_DIS
LIN {X 128.5694,Y 35.0058,Z 152,A 11.38,B 24.8642,C -1.495,E1 25.0607,E2 435.1371} C_DIS
LIN {X 129.9937,Y 29.2716,Z 152,A 8.7072,B 24.8651,C -1.4796,E1 25.0625,E2 437.8306} C_DIS
LIN {X 130.8611,Y 25.108,Z 152,A 6.9829,B 24.8651,C -1.4796,E1 25.0634,E2 439.545} C_DIS
LIN {X 131.4761,Y 21.6597,Z 152,A 5.4089,B 24.8656,C -1.471,E1 25.0641,E2 441.13} C_DIS
LIN {X 132.0902,Y 17.5291,Z 152,A 3.7138,B 24.8656,C -1.4707,E1 25.0648,E2 442.8158} C_DIS
LIN {X 132.4767,Y 14.3173,Z 152,A 2.2711,B 24.866,C -1.4633,E1 25.0653,E2 444.2674} C_DIS
LIN {X 132.8743,Y 9.9789,Z 152,A 0.4321,B 24.8662,C -1.459,E1 25.0657,E2 446.1056} C_DIS
LIN {X 133.0903,Y 6.4883,Z 152,A -1.1077,B 24.8666,C -1.4521,E1 25.0659,E2 447.6526} C_DIS
LIN {X 133.2293,Y 2.246,Z 152,A -2.8592,B 24.8667,C -1.4501,E1 25.066,E2 449.3982} C_DIS
LIN {X 133.231,Y -2.1459,Z 152,A -4.7133,B 24.8669,C -1.4458,E1 25.066,E2 451.2515} C_DIS
LIN {X 133.1198,Y -5.8908,Z 152,A -6.4437,B 24.8676,C -1.4338,E1 25.0658,E2 452.9999} C_DIS
LIN {X 132.8972,Y -9.6645,Z 152,A -7.9516,B 24.8676,C -1.4349,E1 25.0656,E2 454.4961} C_DIS
LIN {X 132.5599,Y -13.5444,Z 152,A -9.7021,B 24.8681,C -1.4252,E1 25.0651,E2 456.2593} C_DIS
LIN {X 132.1178,Y -17.3185,Z 152,A -11.2131,B 24.868,C -1.4266,E1 25.0646,E2 457.7581} C_DIS
LIN {X 131.596,Y -20.9242,Z 152,A -12.902,B 24.8686,C -1.4146,E1 25.0639,E2 459.4652} C_DIS
LIN {X 130.9289,Y -24.7534,Z 152,A -14.4101,B 24.8684,C -1.4181,E1 25.0631,E2 460.9561} C_DIS
LIN {X 130.292,Y -27.9119,Z 152,A -15.8306,B 24.8688,C -1.4117,E1 25.0623,E2 462.3836} C_DIS
LIN {X 129.5112,Y -31.3351,Z 152,A -17.3385,B 24.869,C -1.4068,E1 25.0613,E2 463.8942} C_DIS
LIN {X 128.8291,Y -34.0318,Z 152,A -18.8979,B 24.8703,C -1.3829,E1 25.0602,E2 465.501} C_DIS
LIN {X 127.8121,Y -37.6712,Z 152,A -20.1349,B 24.8695,C -1.399,E1 25.0593,E2 466.6929} C_DIS
LIN {X 126.1617,Y -42.8819,Z 152,A -22.5863,B 24.8701,C -1.3858,E1 25.0571,E2 469.1615} C_DIS
LIN {X 124.8348,Y -46.5968,Z 152,A -24.1393,B 24.8701,C -1.3884,E1 25.0557,E2 470.6998} C_DIS
LIN {X 123.6333,Y -49.6969,Z 152,A -25.5723,B 24.8703,C -1.3837,E1 25.0542,E2 472.136} C_DIS
LIN {X 122.3547,Y -52.7664,Z 152,A -26.9765,B 24.8704,C -1.3806,E1 25.0527,E2 473.5397} C_DIS
LIN {X 120.9985,Y -55.8062,Z 152,A -28.4048,B 24.8706,C -1.3763,E1 25.051,E2 474.9704} C_DIS
LIN {X 119.5797,Y -58.7851,Z 152,A -29.7415,B 24.8706,C -1.3765,E1 25.0494,E2 476.2995} C_DIS
LIN {X 118.0612,Y -61.7781,Z 152,A -31.2445,B 24.871,C -1.3688,E1 25.0475,E2 477.8127} C_DIS
LIN {X 116.0299,Y -65.518,Z 152,A -33.1672,B 24.8716,C -1.3581,E1 25.0448,E2 479.7504} C_DIS
LIN {X 113.7723,Y -69.3648,Z 152,A -35.0769,B 24.8718,C -1.3529,E1 25.0421,E2 481.6627} C_DIS
LIN {X 111.6068,Y -72.7974,Z 152,A -36.8122,B 24.8721,C -1.3484,E1 25.0395,E2 483.3999} C_DIS
LIN {X 109.1184,Y -76.4774,Z 152,A -38.6235,B 24.8721,C -1.3484,E1 25.0366,E2 485.2023} C_DIS
LIN {X 106.7718,Y -79.72,Z 152,A -40.158,B 24.8718,C -1.3538,E1 25.0341,E2 486.7166} C_DIS
LIN {X 104.5714,Y -82.5858,Z 152,A -41.9734,B 24.8727,C -1.3351,E1 25.031,E2 488.5675} C_DIS
LIN {X 101.8064,Y -85.9715,Z 152,A -43.8537,B 24.873,C -1.33,E1 25.0276,E2 490.4512} C_DIS
LIN {X 98.9669,Y -89.2255,Z 152,A -45.6811,B 24.8732,C -1.3268,E1 25.0242,E2 492.2781} C_DIS
LIN {X 95.9597,Y -92.4517,Z 152,A -47.585,B 24.8734,C -1.3215,E1 25.0206,E2 494.1861} C_DIS
LIN {X 92.7373,Y -95.6831,Z 152,A -49.4811,B 24.8734,C -1.3203,E1 25.0168,E2 496.0772} C_DIS
LIN {X 89.5534,Y -98.6694,Z 152,A -51.3741,B 24.8737,C -1.3149,E1 25.0129,E2 497.9753} C_DIS
LIN {X 86.1164,Y -101.6833,Z 152,A -53.3197,B 24.8739,C -1.3113,E1 25.0088,E2 499.9215} C_DIS
LIN {X 82.6764,Y -104.4999,Z 152,A -55.2367,B 24.8741,C -1.3068,E1 25.0046,E2 501.8421} C_DIS
LIN {X 79.1895,Y -107.1663,Z 152,A -57.2425,B 24.8747,C -1.2963,E1 25.0001,E2 503.8655} C_DIS
LIN {X 75.0475,Y -110.1068,Z 152,A -59.286,B 24.8745,C -1.2993,E1 24.9954,E2 505.8947} C_DIS
LIN {X 70.0468,Y -113.3538,Z 152,A -62.4015,B 24.8762,C -1.2647,E1 24.9879,E2 509.0823} C_DIS
LIN {X 65.6048,Y -115.9811,Z 152,A -64.0563,B 24.8749,C -1.2908,E1 24.9841,E2 510.6702} C_DIS
LIN {X 62.1049,Y -117.8896,Z 152,A -65.6738,B 24.8749,C -1.293,E1 24.9801,E2 512.2779} C_DIS
LIN {X 59.0553,Y -119.4463,Z 152,A -67.1142,B 24.8749,C -1.2922,E1 24.9765,E2 513.7161} C_DIS
LIN {X 56.1394,Y -120.8444,Z 152,A -68.5118,B 24.8749,C -1.2896,E1 24.973,E2 515.1164} C_DIS
LIN {X 53.1129,Y -122.2049,Z 152,A -69.9217,B 24.8751,C -1.2883,E1 24.9694,E2 516.526} C_DIS
LIN {X 50.12,Y -123.4628,Z 152,A -71.2988,B 24.8751,C -1.2872,E1 24.9658,E2 517.9024} C_DIS
LIN {X 46.8988,Y -124.7217,Z 152,A -72.7258,B 24.8751,C -1.2883,E1 24.9621,E2 519.3235} C_DIS
LIN {X 43.8923,Y -125.8114,Z 152,A -74.1852,B 24.8754,C -1.282,E1 24.9583,E2 520.795} C_DIS
LIN {X 40.6786,Y -126.8868,Z 152,A -75.6614,B 24.8754,C -1.2792,E1 24.9543,E2 522.2751} C_DIS
LIN {X 36.7047,Y -128.0951,Z 152,A -77.8572,B 24.8766,C -1.2554,E1 24.9483,E2 524.5235} C_DIS
LIN {X 32.9587,Y -129.1076,Z 152,A -79.2005,B 24.8759,C -1.2708,E1 24.9448,E2 525.8282} C_DIS
LIN {X 28.4387,Y -130.1782,Z 152,A -81.1238,B 24.8758,C -1.2728,E1 24.9396,E2 527.744} C_DIS
LIN {X 24.6894,Y -130.9411,Z 152,A -82.7672,B 24.8758,C -1.2715,E1 24.9351,E2 529.3887} C_DIS
LIN {X 20.5428,Y -131.6551,Z 152,A -84.5447,B 24.8758,C -1.2718,E1 24.9302,E2 531.1637} C_DIS
LIN {X 16.5817,Y -132.2144,Z 152,A -86.3645,B 24.8762,C -1.2654,E1 24.9251,E2 532.9972} C_DIS
LIN {X 12.6958,Y -132.6419,Z 152,A -87.92,B 24.8759,C -1.271,E1 24.9208,E2 534.5382} C_DIS
LIN {X 8.9459,Y -132.9496,Z 152,A -89.6659,B 24.8762,C -1.2635,E1 24.9159,E2 536.3012} C_DIS
LIN {X 5.1435,Y -133.1489,Z 152,A -91.1907,B 24.876,C -1.2688,E1 24.9117,E2 537.8129} C_DIS
LIN {X 0.9456,Y -133.2445,Z 152,A -92.926,B 24.8758,C -1.2719,E1 24.9069,E2 539.5405} C_DIS
Enddeposition()
LIN {X 0.9456,Y -133.2445,Z 152,A -92.926,B 24.8758,C -1.2719,E1 24.9069,E2 539.5405} C_DIS
Startdeposition()
$VEL.CP = VEL_PRINT
LIN {X 2.0741,Y -132.2902,Z 152,A -91.4566,B 23.5022,C -1.0596,E1 23.5285,E2 538.4141} C_DIS
LIN {X 5.0048,Y -132.2118,Z 152,A -90.1336,B 23.5022,C -1.0627,E1 23.5322,E2 537.0837} C_DIS
LIN {X 8.883,Y -132.01,Z 152,A -88.333,B 23.5018,C -1.0693,E1 23.5372,E2 535.2675} C_DIS
LIN {X 12.4419,Y -131.7202,Z 152,A -86.9059,B 23.502,C -1.0642,E1 23.5412,E2 533.854} C_DIS
LIN {X 15.7131,Y -131.3699,Z 152,A -85.4826,B 23.502,C -1.0649,E1 23.5451,E2 532.43} C_DIS
LIN {X 19.4795,Y -130.8667,Z 152,A -83.7099,B 23.5017,C -1.0724,E1 23.5501,E2 530.6403} C_DIS
LIN {X 23.0847,Y -130.2769,Z 152,A -82.284,B 23.502,C -1.0658,E1 23.5539,E2 529.2325} C_DIS
LIN {X 27.6972,Y -129.3748,Z 152,A -80.2388,B 23.5019,C -1.068,E1 23.5596,E2 527.1843} C_DIS
LIN {X 30.7801,Y -128.6761,Z 152,A -78.8811,B 23.5019,C -1.0688,E1 23.5632,E2 525.8268} C_DIS
LIN {X 33.8663,Y -127.8985,Z 152,A -77.5041,B 23.5018,C -1.0701,E1 23.567,E2 524.4486} C_DIS
LIN {X 36.9528,Y -127.0411,Z 152,A -76.1184,B 23.5018,C -1.0716,E1 23.5707,E2 523.0618} C_DIS
LIN {X 40.0367,Y -126.1031,Z 152,A -74.7862,B 23.5018,C -1.07,E1 23.5742,E2 521.7361} C_DIS
LIN {X 43.115,Y -125.0841,Z 152,A -73.3056,B 23.5016,C -1.0756,E1 23.5782,E2 520.2446} C_DIS
LIN {X 47.1734,Y -123.6131,Z 152,A -71.3872,B 23.5013,C -1.0806,E1 23.5832,E2 518.3181} C_DIS
LIN {X 50.6175,Y -122.2411,Z 152,A -69.8118,B 23.5013,C -1.0814,E1 23.5873,E2 516.7446} C_DIS
LIN {X 53.737,Y -120.902,Z 152,A -68.375,B 23.5013,C -1.0819,E1 23.591,E2 515.3102} C_DIS
LIN {X 56.757,Y -119.5139,Z 152,A -67.0206,B 23.5013,C -1.0799,E1 23.5944,E2 513.9646} C_DIS
LIN {X 59.2798,Y -118.2854,Z 152,A -65.7398,B 23.5011,C -1.0852,E1 23.5976,E2 512.6742} C_DIS
LIN {X 62.7271,Y -116.4933,Z 152,A -64.0207,B 23.5009,C -1.09,E1 23.6019,E2 510.9484} C_DIS
LIN {X 66.1815,Y -114.5661,Z 152,A -62.2642,B 23.5007,C -1.0953,E1 23.6061,E2 509.1843} C_DIS
LIN {X 70.0077,Y -112.2689,Z 152,A -60.3869,B 23.5007,C -1.0961,E1 23.6106,E2 507.3113} C_DIS
LIN {X 73.6501,Y -109.9139,Z 152,A -58.5268,B 23.5005,C -1.0988,E1 23.6149,E2 505.4508} C_DIS
LIN {X 76.8538,Y -107.698,Z 152,A -56.7861,B 23.5003,C -1.1051,E1 23.6189,E2 503.701} C_DIS
LIN {X 80.2791,Y -105.1696,Z 152,A -54.9501,B 23.5001,C -1.1086,E1 23.623,E2 501.8633} C_DIS
LIN {X 83.8791,Y -102.3215,Z 152,A -53.0333,B 23.5001,C -1.1093,E1 23.6272,E2 499.9523} C_DIS
LIN {X 87.0833,Y -99.6086,Z 152,A -51.2112,B 23.4999,C -1.1137,E1 23.6311,E2 498.1269} C_DIS
LIN {X 90.2584,Y -96.7408,Z 152,A -49.3678,B 23.4997,C -1.1176,E1 23.6349,E2 496.2819} C_DIS
LIN {X 93.341,Y -93.7701,Z 152,A -47.5238,B 23.4995,C -1.1216,E1 23.6385,E2 494.4361} C_DIS
LIN {X 96.1548,Y -90.8825,Z 152,A -45.7381,B 23.4992,C -1.128,E1 23.642,E2 492.6427} C_DIS
LIN {X 99.0435,Y -87.7255,Z 152,A -43.8958,B 23.499,C -1.1322,E1 23.6455,E2 490.7986} C_DIS
LIN {X 101.9918,Y -84.2795,Z 152,A -41.9954,B 23.499,C -1.1341,E1 23.6489,E2 488.9029} C_DIS
LIN {X 104.65,Y -80.9552,Z 152,A -40.1617,B 23.4988,C -1.1385,E1 23.652,E2 487.0673} C_DIS
LIN {X 107.2016,Y -77.5447,Z 152,A -38.3293,B 23.4986,C -1.143,E1 23.6551,E2 485.2332} C_DIS
LIN {X 109.6361,Y -74.0628,Z 152,A -36.5019,B 23.4983,C -1.1475,E1 23.658,E2 483.4042} C_DIS
LIN {X 112.0134,Y -70.416,Z 152,A -34.5756,B 23.498,C -1.155,E1 23.6609,E2 481.4696} C_DIS
LIN {X 114.2938,Y -66.6518,Z 152,A -32.6605,B 23.4977,C -1.1611,E1 23.6636,E2 479.5499} C_DIS
LIN {X 116.3526,Y -62.9889,Z 152,A -30.9338,B 23.4977,C -1.1616,E1 23.6659,E2 477.8315} C_DIS
LIN {X 117.7962,Y -60.2407,Z 152,A -29.6389,B 23.4977,C -1.1631,E1 23.6676,E2 476.5403} C_DIS
LIN {X 119.2861,Y -57.2338,Z 152,A -28.1907,B 23.4974,C -1.1672,E1 23.6694,E2 475.0901} C_DIS
LIN {X 120.6767,Y -54.2407,Z 152,A -26.8242,B 23.4974,C -1.1683,E1 23.6709,E2 473.7289} C_DIS
LIN {X 121.9941,Y -51.2088,Z 152,A -25.3583,B 23.4971,C -1.1745,E1 23.6726,E2 472.2561} C_DIS
LIN {X 123.0189,Y -48.7021,Z 152,A -24.1945,B 23.4969,C -1.1776,E1 23.6738,E2 471.0914} C_DIS
LIN {X 124.2934,Y -45.3462,Z 152,A -22.6196,B 23.4967,C -1.1836,E1 23.6753,E2 469.511} C_DIS
LIN {X 125.4547,Y -42.0244,Z 152,A -21.3609,B 23.4971,C -1.1745,E1 23.6764,E2 468.2826} C_DIS
LIN {X 126.2776,Y -39.4904,Z 152,A -19.9383,B 23.4962,C -1.1922,E1 23.6777,E2 466.8245} C_DIS
LIN {X 127.2012,Y -36.4058,Z 152,A -18.6144,B 23.4962,C -1.1929,E1 23.6787,E2 465.5068} C_DIS
LIN {X 128.0444,Y -33.319,Z 152,A -17.2405,B 23.496,C -1.1968,E1 23.6797,E2 464.1319} C_DIS
LIN {X 128.8479,Y -30.0582,Z 152,A -15.8671,B 23.496,C -1.1972,E1 23.6806,E2 462.7658} C_DIS
LIN {X 129.6037,Y -26.6054,Z 152,A -14.4941,B 23.4962,C -1.1939,E1 23.6814,E2 461.4096} C_DIS
LIN {X 130.2009,Y -23.5096,Z 152,A -12.9346,B 23.4955,C -1.2085,E1 23.6822,E2 459.8235} C_DIS
LIN {X 130.7381,Y -20.3097,Z 152,A -11.5478,B 23.4953,C -1.2121,E1 23.6828,E2 458.4364} C_DIS
LIN {X 131.1554,Y -17.4139,Z 152,A -10.2542,B 23.495,C -1.2176,E1 23.6833,E2 457.1373} C_DIS
LIN {X 131.6283,Y -13.3985,Z 152,A -8.5445,B 23.4948,C -1.2211,E1 23.6838,E2 455.4297} C_DIS
LIN {X 131.9393,Y -9.8513,Z 152,A -6.966,B 23.4945,C -1.2281,E1 23.6842,E2 453.8437} C_DIS
LIN {X 132.1526,Y -6.3819,Z 152,A -5.4702,B 23.4943,C -1.2325,E1 23.6844,E2 452.3465} C_DIS
LIN {X 132.2806,Y -2.6559,Z 152,A -3.8294,B 23.494,C -1.2392,E1 23.6845,E2 450.6996} C_DIS
LIN {X 132.2917,Y 1.9869,Z 152,A -1.9446,B 23.494,C -1.2392,E1 23.6845,E2 448.8269} C_DIS
LIN {X 132.2143,Y 4.9406,Z 152,A -0.6416,B 23.4937,C -1.2445,E1 23.6844,E2 447.5188} C_DIS
LIN {X 132.0583,Y 8.0974,Z 152,A 0.7508,B 23.4934,C -1.2502,E1 23.6842,E2 446.121} C_DIS
LIN {X 131.7688,Y 11.9352,Z 152,A 2.3463,B 23.4934,C -1.2518,E1 23.6838,E2 444.5316} C_DIS
LIN {X 131.4011,Y 15.4512,Z 152,A 3.6786,B 23.4936,C -1.2464,E1 23.6834,E2 443.2212} C_DIS
LIN {X 131.0074,Y 18.4947,Z 152,A 5.2354,B 23.4928,C -1.2626,E1 23.6828,E2 441.6341} C_DIS
LIN {X 130.5129,Y 21.7099,Z 152,A 6.6355,B 23.4926,C -1.2666,E1 23.6822,E2 440.2327} C_DIS
LIN {X 129.8058,Y 25.6121,Z 152,A 8.4761,B 23.492,C -1.2784,E1 23.6812,E2 438.374} C_DIS
LIN {X 129.0353,Y 29.2381,Z 152,A 9.915,B 23.4922,C -1.2748,E1 23.6804,E2 436.9532} C_DIS
LIN {X 128.2972,Y 32.323,Z 152,A 11.2813,B 23.492,C -1.2787,E1 23.6795,E2 435.5856} C_DIS
LIN {X 127.4798,Y 35.4097,Z 152,A 12.6566,B 23.4918,C -1.2826,E1 23.6785,E2 434.209} C_DIS
LIN {X 126.5822,Y 38.4952,Z 152,A 14.0406,B 23.4916,C -1.2865,E1 23.6774,E2 432.8239} C_DIS
LIN {X 125.5808,Y 41.6456,Z 152,A 15.4469,B 23.4914,C -1.2895,E1 23.6762,E2 431.4185} C_DIS
LIN {X 124.5281,Y 44.6951,Z 152,A 16.7785,B 23.4914,C -1.2903,E1 23.6749,E2 430.093} C_DIS
LIN {X 123.4024,Y 47.7154,Z 152,A 18.1861,B 23.4911,C -1.2951,E1 23.6735,E2 428.6818} C_DIS
LIN {X 122.2,Y 50.7159,Z 152,A 19.6483,B 23.4907,C -1.3024,E1 23.672,E2 427.21} C_DIS
LIN {X 120.9802,Y 53.5621,Z 152,A 20.8429,B 23.4909,C -1.2987,E1 23.6707,E2 426.0316} C_DIS
LIN {X 119.7402,Y 56.2835,Z 152,A 22.2561,B 23.4904,C -1.3086,E1 23.669,E2 424.602} C_DIS
LIN {X 118.2854,Y 59.2798,Z 152,A 23.6907,B 23.4902,C -1.3122,E1 23.6672,E2 423.1665} C_DIS
LIN {X 116.4336,Y 62.8382,Z 152,A 25.4396,B 23.4899,C -1.3177,E1 23.6649,E2 421.4138} C_DIS
LIN {X 114.5661,Y 66.1815,Z 152,A 27.1586,B 23.4895,C -1.3254,E1 23.6625,E2 419.6852} C_DIS
LIN {X 112.2689,Y 70.0077,Z 152,A 29.0575,B 23.4893,C -1.3288,E1 23.6598,E2 417.7882} C_DIS
LIN {X 109.9717,Y 73.5636,Z 152,A 30.8564,B 23.4892,C -1.3318,E1 23.657,E2 415.9913} C_DIS
LIN {X 107.698,Y 76.8538,Z 152,A 32.6288,B 23.4888,C -1.3383,E1 23.6542,E2 414.212} C_DIS
LIN {X 105.1236,Y 80.3392,Z 152,A 34.4798,B 23.4886,C -1.3417,E1 23.6511,E2 412.3621} C_DIS
LIN {X 102.3692,Y 83.8207,Z 152,A 36.3594,B 23.4886,C -1.3441,E1 23.6478,E2 410.4857} C_DIS
LIN {X 99.5687,Y 87.129,Z 152,A 38.2169,B 23.4883,C -1.3475,E1 23.6444,E2 408.6287} C_DIS
LIN {X 96.7408,Y 90.2584,Z 152,A 40.0497,B 23.4881,C -1.352,E1 23.6409,E2 406.7934} C_DIS
LIN {X 93.7644,Y 93.3466,Z 152,A 41.8918,B 23.4879,C -1.3553,E1 23.6373,E2 404.9515} C_DIS
LIN {X 90.8825,Y 96.1548,Z 152,A 43.6771,B 23.4876,C -1.3612,E1 23.6337,E2 403.1595} C_DIS
LIN {X 87.5013,Y 99.2417,Z 152,A 45.5924,B 23.4876,C -1.3618,E1 23.6298,E2 401.2509} C_DIS
LIN {X 84.4799,Y 101.8259,Z 152,A 47.364,B 23.4872,C -1.3677,E1 23.626,E2 399.4718} C_DIS
LIN {X 80.9552,Y 104.65,Z 152,A 49.2618,B 23.4872,C -1.3684,E1 23.6218,E2 397.5799} C_DIS
LIN {X 77.5447,Y 107.2016,Z 152,A 51.0981,B 23.487,C -1.3712,E1 23.6177,E2 395.7434} C_DIS
LIN {X 74.0628,Y 109.6361,Z 152,A 52.9459,B 23.4868,C -1.3748,E1 23.6134,E2 393.8936} C_DIS
LIN {X 70.5157,Y 111.9505,Z 152,A 54.7564,B 23.4868,C -1.3765,E1 23.6092,E2 392.085} C_DIS
LIN {X 66.8121,Y 114.1996,Z 152,A 56.6801,B 23.4865,C -1.3817,E1 23.6045,E2 390.1547} C_DIS
LIN {X 62.9889,Y 116.3526,Z 152,A 58.549,B 23.4864,C -1.3828,E1 23.6,E2 388.2888} C_DIS
LIN {X 60.2407,Y 117.7962,Z 152,A 59.815,B 23.4865,C -1.3807,E1 23.5969,E2 387.0318} C_DIS
LIN {X 57.2524,Y 119.2773,Z 152,A 61.2538,B 23.4865,C -1.3823,E1 23.5932,E2 385.5932} C_DIS
LIN {X 54.2407,Y 120.6767,Z 152,A 62.693,B 23.4863,C -1.384,E1 23.5896,E2 384.1536} C_DIS
LIN {X 51.2088,Y 121.9941,Z 152,A 64.1134,B 23.4863,C -1.3851,E1 23.5859,E2 382.7341} C_DIS
LIN {X 48.7021,Y 123.0189,Z 152,A 65.2826,B 23.4863,C -1.3861,E1 23.5829,E2 381.5653} C_DIS
LIN {X 45.3022,Y 124.3092,Z 152,A 66.9016,B 23.486,C -1.3898,E1 23.5787,E2 379.9406} C_DIS
LIN {X 42.0244,Y 125.4547,Z 152,A 68.1297,B 23.4867,C -1.3776,E1 23.5755,E2 378.7458} C_DIS
LIN {X 39.4904,Y 126.2776,Z 152,A 69.5011,B 23.486,C -1.3892,E1 23.5718,E2 377.348} C_DIS
LIN {X 36.4058,Y 127.2012,Z 152,A 71.0478,B 23.4856,C -1.3977,E1 23.5676,E2 375.7828} C_DIS
LIN {X 32.7896,Y 128.1788,Z 152,A 72.2984,B 23.4865,C -1.3805,E1 23.5643,E2 374.5772} C_DIS
LIN {X 30.2332,Y 128.808,Z 152,A 73.7754,B 23.4856,C -1.3977,E1 23.5602,E2 373.0596} C_DIS
LIN {X 26.6054,Y 129.6037,Z 152,A 75.0354,B 23.4865,C -1.3815,E1 23.5569,E2 371.8419} C_DIS
LIN {X 23.5221,Y 130.1986,Z 152,A 76.6219,B 23.4858,C -1.3931,E1 23.5525,E2 370.2283} C_DIS
LIN {X 20.2459,Y 130.748,Z 152,A 78.0057,B 23.4859,C -1.3909,E1 23.5487,E2 368.8514} C_DIS
LIN {X 16.4313,Y 131.2842,Z 152,A 79.8596,B 23.4854,C -1.4003,E1 23.5435,E2 366.9755} C_DIS
LIN {X 12.6634,Y 131.6989,Z 152,A 81.384,B 23.4857,C -1.3949,E1 23.5393,E2 365.4657} C_DIS
LIN {X 8.8025,Y 132.0149,Z 152,A 83.1449,B 23.4855,C -1.399,E1 23.5343,E2 363.6955} C_DIS
LIN {X 5.257,Y 132.202,Z 152,A 84.5248,B 23.4859,C -1.3914,E1 23.5306,E2 362.3352} C_DIS
LIN {X 2.1125,Y 132.2896,Z 152,A 85.9881,B 23.4856,C -1.3961,E1 23.5264,E2 360.8603} C_DIS
LIN {X -1.9869,Y 132.2917,Z 152,A 87.7232,B 23.4858,C -1.3938,E1 23.5216,E2 359.131} C_DIS
LIN {X -5.2993,Y 132.2003,Z 152,A 89.1959,B 23.4857,C -1.3952,E1 23.5175,E2 357.6546} C_DIS
LIN {X -8.9168,Y 132.0075,Z 152,A 90.8443,B 23.4855,C -1.3984,E1 23.5129,E2 355.9975} C_DIS
LIN {X -13.3985,Y 131.6283,Z 152,A 92.8103,B 23.4855,C -1.3984,E1 23.5074,E2 354.0307} C_DIS
LIN {X -17.126,Y 131.1932,Z 152,A 94.3042,B 23.4859,C -1.3911,E1 23.5033,E2 352.5537} C_DIS
LIN {X -20.4665,Y 130.7138,Z 152,A 95.8078,B 23.4859,C -1.3922,E1 23.4991,E2 351.0461} C_DIS
LIN {X -24.6202,Y 129.9955,Z 152,A 97.3683,B 23.4866,C -1.3782,E1 23.4949,E2 349.5189} C_DIS
LIN {X -27.6972,Y 129.3748,Z 152,A 98.9479,B 23.4861,C -1.3875,E1 23.4906,E2 347.914} C_DIS
LIN {X -30.7801,Y 128.6761,Z 152,A 100.3353,B 23.4861,C -1.3871,E1 23.4868,E2 346.5256} C_DIS
LIN {X -34.0041,Y 127.8617,Z 152,A 101.7334,B 23.4863,C -1.3837,E1 23.483,E2 345.1338} C_DIS
LIN {X -36.9528,Y 127.0411,Z 152,A 103.0976,B 23.4863,C -1.3842,E1 23.4793,E2 343.7663} C_DIS
LIN {X -40.0416,Y 126.1016,Z 152,A 104.4362,B 23.4866,C -1.3798,E1 23.4758,E2 342.4362} C_DIS
LIN {X -43.115,Y 125.0841,Z 152,A 105.9085,B 23.4865,C -1.3814,E1 23.4719,E2 340.9569} C_DIS
LIN {X -45.6417,Y 124.1869,Z 152,A 107.224,B 23.4862,C -1.3871,E1 23.4684,E2 339.6242} C_DIS
LIN {X -48.707,Y 123.0169,Z 152,A 108.4992,B 23.4866,C -1.3783,E1 23.4651,E2 338.3681} C_DIS
LIN {X -51.7481,Y 121.7689,Z 152,A 109.931,B 23.4867,C -1.3767,E1 23.4614,E2 336.9369} C_DIS
LIN {X -54.7767,Y 120.4369,Z 152,A 111.5102,B 23.4865,C -1.3814,E1 23.4574,E2 335.3417} C_DIS
LIN {X -57.7846,Y 119.023,Z 152,A 112.8157,B 23.4869,C -1.3729,E1 23.4541,E2 334.0541} C_DIS
LIN {X -60.7686,Y 117.5275,Z 152,A 114.3868,B 23.4867,C -1.3764,E1 23.4502,E2 332.4696} C_DIS
LIN {X -64.5713,Y 115.4816,Z 152,A 116.2734,B 23.4869,C -1.3739,E1 23.4456,E2 330.5835} C_DIS
LIN {X -68.5686,Y 113.1535,Z 152,A 118.2469,B 23.4872,C -1.3689,E1 23.4408,E2 328.6162} C_DIS
LIN {X -72.2536,Y 110.837,Z 152,A 120.1504,B 23.4873,C -1.3662,E1 23.4364,E2 326.713} C_DIS
LIN {X -75.9139,Y 108.3634,Z 152,A 122.0513,B 23.4875,C -1.3618,E1 23.432,E2 324.8163} C_DIS
LIN {X -79.3587,Y 105.8665,Z 152,A 123.9587,B 23.4875,C -1.361,E1 23.4277,E2 322.9037} C_DIS
LIN {X -82.7291,Y 103.2542,Z 152,A 125.8165,B 23.4878,C -1.3575,E1 23.4236,E2 321.0473} C_DIS
LIN {X -86.1528,Y 100.4147,Z 152,A 127.6985,B 23.4881,C -1.3511,E1 23.4196,E2 319.1735} C_DIS
LIN {X -89.2239,Y 97.6966,Z 152,A 129.5284,B 23.4882,C -1.3495,E1 23.4158,E2 317.3399} C_DIS
LIN {X -92.3374,Y 94.7593,Z 152,A 131.3921,B 23.4884,C -1.3455,E1 23.4121,E2 315.4778} C_DIS
LIN {X -95.4589,Y 91.6135,Z 152,A 133.2364,B 23.4889,C -1.3374,E1 23.4085,E2 313.6457} C_DIS
LIN {X -98.2717,Y 88.5901,Z 152,A 135.1083,B 23.4889,C -1.3367,E1 23.405,E2 311.7666} C_DIS
LIN {X -101.0833,Y 85.368,Z 152,A 136.9713,B 23.4891,C -1.3324,E1 23.4016,E2 309.9053} C_DIS
LIN {X -103.7857,Y 82.0613,Z 152,A 138.8419,B 23.4893,C -1.3285,E1 23.3983,E2 308.0353} C_DIS
LIN {X -106.3753,Y 78.6755,Z 152,A 140.6981,B 23.4896,C -1.324,E1 23.3952,E2 306.1809} C_DIS
LIN {X -108.8935,Y 75.1511,Z 152,A 142.5443,B 23.4899,C -1.3174,E1 23.3923,E2 304.3415} C_DIS
LIN {X -111.2028,Y 71.6901,Z 152,A 144.4014,B 23.4901,C -1.3148,E1 23.3894,E2 302.4809} C_DIS
LIN {X -113.5233,Y 67.955,Z 152,A 146.3121,B 23.4903,C -1.3097,E1 23.3867,E2 300.5728} C_DIS
LIN {X -115.6884,Y 64.1995,Z 152,A 148.1705,B 23.4907,C -1.3033,E1 23.3841,E2 298.7199} C_DIS
LIN {X -117.5275,Y 60.7686,Z 152,A 149.7751,B 23.4911,C -1.2946,E1 23.382,E2 297.128} C_DIS
LIN {X -119.1029,Y 57.6173,Z 152,A 151.2376,B 23.4915,C -1.2872,E1 23.3802,E2 295.6759} C_DIS
LIN {X -120.598,Y 54.4164,Z 152,A 152.6952,B 23.4919,C -1.2793,E1 23.3786,E2 294.2296} C_DIS
LIN {X -121.7689,Y 51.7481,Z 152,A 154.1179,B 23.4917,C -1.2827,E1 23.377,E2 292.79} C_DIS
LIN {X -123.1517,Y 48.3605,Z 152,A 155.7686,B 23.4918,C -1.2808,E1 23.3752,E2 291.1342} C_DIS
LIN {X -124.383,Y 45.0976,Z 152,A 157.2485,B 23.4922,C -1.2748,E1 23.3738,E2 289.6606} C_DIS
LIN {X -125.4703,Y 41.9777,Z 152,A 158.6666,B 23.4924,C -1.2697,E1 23.3725,E2 288.2466} C_DIS
LIN {X -126.4205,Y 39.0236,Z 152,A 159.9958,B 23.4927,C -1.2648,E1 23.3714,E2 286.9216} C_DIS
LIN {X -127.2982,Y 36.059,Z 152,A 161.2281,B 23.4931,C -1.2557,E1 23.3705,E2 285.7046} C_DIS
LIN {X -128.0444,Y 33.319,Z 152,A 162.7009,B 23.4928,C -1.2627,E1 23.3694,E2 284.2049} C_DIS
LIN {X -128.899,Y 29.8345,Z 152,A 164.0088,B 23.4936,C -1.2467,E1 23.3686,E2 282.9293} C_DIS
LIN {X -129.6037,Y 26.6054,Z 152,A 165.3906,B 23.4939,C -1.2399,E1 23.3678,E2 281.5559} C_DIS
LIN {X -130.0996,Y 24.0753,Z 152,A 166.7299,B 23.4936,C -1.2462,E1 23.3671,E2 280.1921} C_DIS
LIN {X -130.7138,Y 20.4665,Z 152,A 168.3582,B 23.4938,C -1.2431,E1 23.3663,E2 278.5614} C_DIS
LIN {X -131.1554,Y 17.4139,Z 152,A 169.6242,B 23.4941,C -1.2356,E1 23.3658,E2 277.3061} C_DIS
LIN {X -131.6283,Y 13.3985,Z 152,A 171.4276,B 23.4943,C -1.2322,E1 23.3653,E2 275.4997} C_DIS
LIN {X -131.9393,Y 9.8513,Z 152,A 173.0123,B 23.4944,C -1.2292,E1 23.3649,E2 273.9126} C_DIS
LIN {X -132.1498,Y 6.4379,Z 152,A 174.5225,B 23.4946,C -1.2257,E1 23.3647,E2 272.4014} C_DIS
LIN {X -132.2759,Y 2.9367,Z 152,A 175.9923,B 23.495,C -1.2186,E1 23.3646,E2 270.94} C_DIS
LIN {X -132.3067,Y -0.5353,Z 152,A 177.5461,B 23.495,C -1.2159,E1 23.3646,E2 269.3829} C_DIS
LIN {X -132.2143,Y -4.9406,Z 152,A 179.4713,B 23.4954,C -1.2105,E1 23.3647,E2 267.4589} C_DIS
LIN {X -132.048,Y -8.2656,Z 152,A -179.0416,B 23.4954,C -1.2079,E1 23.3649,E2 265.9688} C_DIS
LIN {X -131.7219,Y -12.4239,Z 152,A -177.4992,B 23.4963,C -1.1902,E1 23.3653,E2 264.4612} C_DIS
LIN {X -131.4011,Y -15.4512,Z 152,A -175.9969,B 23.4961,C -1.1943,E1 23.3658,E2 262.939} C_DIS
LIN {X -130.8667,Y -19.4795,Z 152,A -174.0255,B 23.496,C -1.1982,E1 23.3665,E2 260.945} C_DIS
LIN {X -130.2769,Y -23.0847,Z 152,A -172.5872,B 23.4965,C -1.1867,E1 23.3672,E2 259.5266} C_DIS
LIN {X -129.3748,Y -27.6972,Z 152,A -170.5342,B 23.4968,C -1.1811,E1 23.3683,E2 257.4748} C_DIS
LIN {X -128.6761,Y -30.7801,Z 152,A -169.1478,B 23.4969,C -1.1776,E1 23.3692,E2 256.0884} C_DIS
LIN {X -127.8985,Y -33.8663,Z 152,A -167.7636,B 23.4971,C -1.1736,E1 23.3702,E2 254.7057} C_DIS
LIN {X -127.0117,Y -37.053,Z 152,A -166.3445,B 23.4974,C -1.1686,E1 23.3713,E2 253.2904} C_DIS
LIN {X -126.0981,Y -40.0525,Z 152,A -164.9837,B 23.4976,C -1.1646,E1 23.3724,E2 251.9313} C_DIS
LIN {X -125.0841,Y -43.115,Z 152,A -163.7666,B 23.4981,C -1.1522,E1 23.3735,E2 250.7381} C_DIS
LIN {X -124.1869,Y -45.6417,Z 152,A -162.3718,B 23.4978,C -1.1593,E1 23.3748,E2 249.3168} C_DIS
LIN {X -122.8459,Y -49.1311,Z 152,A -160.727,B 23.498,C -1.1558,E1 23.3765,E2 247.6711} C_DIS
LIN {X -121.5364,Y -52.2859,Z 152,A -159.4777,B 23.4986,C -1.141,E1 23.3778,E2 246.4517} C_DIS
LIN {X -120.4369,Y -54.7767,Z 152,A -158.0617,B 23.4983,C -1.1483,E1 23.3794,E2 245.0089} C_DIS
LIN {X -118.8582,Y -58.1187,Z 152,A -156.5007,B 23.4986,C -1.142,E1 23.3813,E2 243.4547} C_DIS
LIN {X -117.2874,Y -61.2257,Z 152,A -154.9267,B 23.4986,C -1.1408,E1 23.3833,E2 241.8746} C_DIS
LIN {X -115.2784,Y -64.9328,Z 152,A -153.0223,B 23.4987,C -1.1394,E1 23.3859,E2 239.9631} C_DIS
LIN {X -113.0847,Y -68.6825,Z 152,A -151.1028,B 23.4989,C -1.1361,E1 23.3887,E2 238.0413} C_DIS
LIN {X -110.7416,Y -72.4005,Z 152,A -149.1619,B 23.499,C -1.1328,E1 23.3916,E2 236.0982} C_DIS
LIN {X -108.2812,Y -76.0304,Z 152,A -147.283,B 23.4993,C -1.1271,E1 23.3946,E2 234.2239} C_DIS
LIN {X -105.8665,Y -79.3587,Z 152,A -145.505,B 23.4995,C -1.1225,E1 23.3975,E2 232.4482} C_DIS
LIN {X -103.2542,Y -82.7291,Z 152,A -143.5894,B 23.4995,C -1.1212,E1 23.4008,E2 230.5261} C_DIS
LIN {X -100.4431,Y -86.1198,Z 152,A -141.6987,B 23.4998,C -1.116,E1 23.4042,E2 228.6394} C_DIS
LIN {X -97.5699,Y -89.3617,Z 152,A -139.809,B 23.4999,C -1.1123,E1 23.4078,E2 226.7498} C_DIS
LIN {X -94.7593,Y -92.3374,Z 152,A -138.0156,B 23.5001,C -1.1094,E1 23.4112,E2 224.9555} C_DIS
LIN {X -91.7223,Y -95.3549,Z 152,A -136.1447,B 23.5002,C -1.1063,E1 23.415,E2 223.0841} C_DIS
LIN {X -88.5901,Y -98.2717,Z 152,A -134.3376,B 23.5005,C -1.1003,E1 23.4187,E2 221.2842} C_DIS
LIN {X -85.368,Y -101.0833,Z 152,A -132.4627,B 23.5005,C -1.0978,E1 23.4227,E2 219.4079} C_DIS
LIN {X -82.0243,Y -103.8148,Z 152,A -130.5669,B 23.5007,C -1.0955,E1 23.4268,E2 217.5103} C_DIS
LIN {X -78.6755,Y -106.3753,Z 152,A -128.7229,B 23.5007,C -1.0931,E1 23.4309,E2 215.6651} C_DIS
LIN {X -75.2165,Y -108.8486,Z 152,A -126.8602,B 23.5009,C -1.091,E1 23.4352,E2 213.801} C_DIS
LIN {X -71.6875,Y -111.2045,Z 152,A -125.0687,B 23.5011,C -1.0859,E1 23.4394,E2 212.0161} C_DIS
LIN {X -68.1025,Y -113.4353,Z 152,A -123.1804,B 23.5011,C -1.0859,E1 23.4439,E2 210.1212} C_DIS
LIN {X -64.1995,Y -115.6884,Z 152,A -121.2722,B 23.5013,C -1.0812,E1 23.4485,E2 208.2192} C_DIS
LIN {X -60.4087,Y -117.7107,Z 152,A -119.6543,B 23.5019,C -1.0672,E1 23.4524,E2 206.6317} C_DIS
LIN {X -57.4313,Y -119.1918,Z 152,A -118.0837,B 23.5017,C -1.0716,E1 23.4564,E2 205.0456} C_DIS
LIN {X -54.393,Y -120.6085,Z 152,A -116.5779,B 23.5017,C -1.0725,E1 23.4602,E2 203.5336} C_DIS
LIN {X -51.2088,Y -121.9941,Z 152,A -115.0958,B 23.5018,C -1.0698,E1 23.464,E2 202.0545} C_DIS
LIN {X -48.1183,Y -123.2458,Z 152,A -113.6397,B 23.5018,C -1.069,E1 23.4678,E2 200.5971} C_DIS
LIN {X -44.1071,Y -124.7401,Z 152,A -111.7947,B 23.5019,C -1.0668,E1 23.4726,E2 198.7535} C_DIS
LIN {X -41.0311,Y -125.7855,Z 152,A -110.387,B 23.5019,C -1.0657,E1 23.4764,E2 197.3458} C_DIS
LIN {X -37.4575,Y -126.8933,Z 152,A -108.7939,B 23.5021,C -1.0632,E1 23.4806,E2 195.756} C_DIS
LIN {X -34.4348,Y -127.7469,Z 152,A -107.5767,B 23.5024,C -1.0554,E1 23.4839,E2 194.5564} C_DIS
LIN {X -31.3354,Y -128.5423,Z 152,A -106.1952,B 23.5024,C -1.0544,E1 23.4876,E2 193.1753} C_DIS
LIN {X -28.6914,Y -129.1601,Z 152,A -104.6865,B 23.5018,C -1.0699,E1 23.4918,E2 191.6256} C_DIS
LIN {X -25.0071,Y -129.9215,Z 152,A -103.2339,B 23.5022,C -1.0607,E1 23.4957,E2 190.1944} C_DIS
LIN {X -21.8313,Y -130.4926,Z 152,A -101.8604,B 23.5022,C -1.0591,E1 23.4995,E2 188.8236} C_DIS
LIN {X -17.4139,Y -131.1554,Z 152,A -99.8542,B 23.5022,C -1.0621,E1 23.5051,E2 186.8081} C_DIS
LIN {X -14.3759,Y -131.5231,Z 152,A -98.5241,B 23.5022,C -1.0621,E1 23.5088,E2 185.477} C_DIS
LIN {X -10.9169,Y -131.8553,Z 152,A -97.0057,B 23.5022,C -1.0627,E1 23.513,E2 183.9564} C_DIS
LIN {X -6.8598,Y -132.1286,Z 152,A -95.3018,B 23.5022,C -1.0599,E1 23.5177,E2 182.2588} C_DIS
LIN {X -3.8286,Y -132.2511,Z 152,A -93.9354,B 23.5022,C -1.0626,E1 23.5216,E2 180.8853} C_DIS
LIN {X 0,Y -132.3085,Z 152,A -92.1727,B 23.5019,C -1.0681,E1 23.5265,E2 179.1089} C_DIS
LIN {X 0,Y -132.3085,Z 152,A -92.1727,B 23.5019,C -1.0681,E1 23.5265,E2 179.1089} C_DIS
Enddeposition()
LIN {X 0.9353,Y -131.3597,Z 152,A -92.1346,B 22.3979,C -0.86,E1 22.4143,E2 179.4713} C_DIS
Startdeposition()
$VEL.CP = VEL_PRINT
LIN {X -2.3928,Y -131.343,Z 152,A -93.7287,B 22.3981,C -0.8532,E1 22.4098,E2 181.0833} C_DIS
LIN {X -6.5451,Y -131.2014,Z 152,A -95.574,B 22.3981,C -0.8515,E1 22.4046,E2 182.9334} C_DIS
LIN {X -10.8461,Y -130.9161,Z 152,A -97.3762,B 22.3981,C -0.8551,E1 22.3996,E2 184.7269} C_DIS
LIN {X -14.467,Y -130.5661,Z 152,A -99.0383,B 22.3981,C -0.8519,E1 22.395,E2 186.3986} C_DIS
LIN {X -19.1476,Y -129.9627,Z 152,A -100.9428,B 22.3979,C -0.8593,E1 22.3897,E2 188.2852} C_DIS
LIN {X -22.7239,Y -129.3847,Z 152,A -102.5899,B 22.3979,C -0.8568,E1 22.3852,E2 189.9407} C_DIS
LIN {X -26.0191,Y -128.7619,Z 152,A -103.9405,B 22.3978,C -0.8625,E1 22.3815,E2 191.278} C_DIS
LIN {X -30.5338,Y -127.7667,Z 152,A -105.8327,B 22.3975,C -0.8691,E1 22.3764,E2 193.1555} C_DIS
LIN {X -34.7457,Y -126.6875,Z 152,A -108.0579,B 22.398,C -0.8554,E1 22.3703,E2 195.4205} C_DIS
LIN {X -38.2734,Y -125.6651,Z 152,A -109.6328,B 22.398,C -0.8578,E1 22.3661,E2 196.9921} C_DIS
LIN {X -42.1708,Y -124.4133,Z 152,A -111.4677,B 22.398,C -0.857,E1 22.3612,E2 198.8329} C_DIS
LIN {X -45.9053,Y -123.0824,Z 152,A -113.0274,B 22.3976,C -0.8661,E1 22.3571,E2 200.3721} C_DIS
LIN {X -48.7587,Y -121.9806,Z 152,A -114.4288,B 22.3977,C -0.8644,E1 22.3535,E2 201.7813} C_DIS
LIN {X -52.9109,Y -120.2397,Z 152,A -116.5061,B 22.3978,C -0.8615,E1 22.3481,E2 203.872} C_DIS
LIN {X -56.4048,Y -118.6384,Z 152,A -118.0853,B 22.3976,C -0.8678,E1 22.3441,E2 205.439} C_DIS
LIN {X -60.2699,Y -116.7245,Z 152,A -120.104,B 22.3977,C -0.864,E1 22.3391,E2 207.4737} C_DIS
LIN {X -64.3996,Y -114.4977,Z 152,A -122.0668,B 22.3975,C -0.8705,E1 22.3343,E2 209.4257} C_DIS
LIN {X -68.2068,Y -112.2716,Z 152,A -124.2013,B 22.3977,C -0.8641,E1 22.3291,E2 211.5845} C_DIS
LIN {X -72.5682,Y -109.5036,Z 152,A -126.3048,B 22.3974,C -0.8742,E1 22.3242,E2 213.6692} C_DIS
LIN {X -75.0475,Y -107.8188,Z 152,A -127.7112,B 22.3974,C -0.872,E1 22.321,E2 215.0866} C_DIS
LIN {X -78.9393,Y -105.0031,Z 152,A -129.7324,B 22.3972,C -0.8789,E1 22.3165,E2 217.0978} C_DIS
LIN {X -82.5046,Y -102.2253,Z 152,A -131.6551,B 22.397,C -0.8846,E1 22.3123,E2 219.0134} C_DIS
LIN {X -85.8247,Y -99.4543,Z 152,A -133.5828,B 22.3969,C -0.8865,E1 22.3082,E2 220.9448} C_DIS
LIN {X -88.9076,Y -96.7081,Z 152,A -135.485,B 22.3969,C -0.8857,E1 22.3042,E2 222.8576} C_DIS
LIN {X -92.382,Y -93.3952,Z 152,A -137.5072,B 22.3966,C -0.8932,E1 22.3002,E2 224.8696} C_DIS
LIN {X -95.3157,Y -90.3994,Z 152,A -139.3627,B 22.3966,C -0.896,E1 22.2966,E2 226.7268} C_DIS
LIN {X -98.3133,Y -87.1295,Z 152,A -141.2989,B 22.3964,C -0.9003,E1 22.293,E2 228.6613} C_DIS
LIN {X -101.2986,Y -83.64,Z 152,A -143.3035,B 22.3962,C -0.9049,E1 22.2894,E2 230.6642} C_DIS
LIN {X -103.9285,Y -80.3487,Z 152,A -145.1218,B 22.396,C -0.9101,E1 22.2862,E2 232.4784} C_DIS
LIN {X -106.5895,Y -76.7843,Z 152,A -147.1056,B 22.3959,C -0.913,E1 22.2829,E2 234.4654} C_DIS
LIN {X -108.9106,Y -73.4544,Z 152,A -148.8789,B 22.3957,C -0.9174,E1 22.2801,E2 236.237} C_DIS
LIN {X -110.4697,Y -71.0885,Z 152,A -150.3542,B 22.396,C -0.9104,E1 22.2779,E2 237.7392} C_DIS
LIN {X -112.3359,Y -68.1006,Z 152,A -152.7819,B 22.3972,C -0.8771,E1 22.2743,E2 240.2691} C_DIS
LIN {X -116.1621,Y -61.343,Z 152,A -155.003,B 22.395,C -0.9353,E1 22.2715,E2 242.3498} C_DIS
LIN {X -117.701,Y -58.3356,Z 152,A -156.4763,B 22.3948,C -0.9394,E1 22.2696,E2 243.8212} C_DIS
LIN {X -119.0192,Y -55.5987,Z 152,A -157.6723,B 22.3945,C -0.9486,E1 22.2682,E2 245.0002} C_DIS
LIN {X -120.9593,Y -51.2426,Z 152,A -159.8285,B 22.3944,C -0.9513,E1 22.2658,E2 247.1628} C_DIS
LIN {X -124.0276,Y -43.287,Z 152,A -163.7878,B 22.3944,C -0.952,E1 22.2619,E2 251.1454} C_DIS
LIN {X -125.4528,Y -38.9671,Z 152,A -165.6865,B 22.394,C -0.9616,E1 22.2602,E2 253.0311} C_DIS
LIN {X -126.4611,Y -35.5554,Z 152,A -167.2114,B 22.3937,C -0.9674,E1 22.2591,E2 254.5506} C_DIS
LIN {X -127.3065,Y -32.3981,Z 152,A -168.6474,B 22.3936,C -0.9713,E1 22.258,E2 255.9857} C_DIS
LIN {X -128.1196,Y -29.0174,Z 152,A -170.2034,B 22.3934,C -0.9744,E1 22.2571,E2 257.5441} C_DIS
LIN {X -128.9123,Y -25.2703,Z 152,A -171.9379,B 22.3934,C -0.9768,E1 22.2561,E2 259.2836} C_DIS
LIN {X -129.6186,Y -21.3472,Z 152,A -173.611,B 22.393,C -0.9851,E1 22.2553,E2 260.9462} C_DIS
LIN {X -130.2525,Y -17.0555,Z 152,A -176.6521,B 22.3947,C -0.9434,E1 22.2542,E2 264.1179} C_DIS
LIN {X -131.0144,Y -9.5848,Z 152,A -178.8568,B 22.3924,C -0.9981,E1 22.2537,E2 266.193} C_DIS
LIN {X -131.327,Y -3.1778,Z 152,A 178.1857,B 22.3924,C -1.0004,E1 22.2533,E2 269.1647} C_DIS
LIN {X -131.2362,Y 5.8519,Z 152,A 174.2726,B 22.3918,C -1.0141,E1 22.2536,E2 273.0682} C_DIS
LIN {X -131.0098,Y 9.6469,Z 152,A 172.5582,B 22.3916,C -1.0171,E1 22.2539,E2 274.7863} C_DIS
LIN {X -130.2892,Y 16.7755,Z 152,A 169.5715,B 22.3909,C -1.0329,E1 22.2548,E2 277.7515} C_DIS
LIN {X -129.8069,Y 20.1687,Z 152,A 168.0436,B 22.3908,C -1.0363,E1 22.2554,E2 279.2807} C_DIS
LIN {X -129.1732,Y 23.9047,Z 152,A 166.2891,B 22.3908,C -1.0373,E1 22.2563,E2 281.0443} C_DIS
LIN {X -128.4308,Y 27.6066,Z 152,A 164.703,B 22.3904,C -1.0451,E1 22.2572,E2 282.6204} C_DIS
LIN {X -127.4843,Y 31.6973,Z 152,A 162.9414,B 22.39,C -1.0538,E1 22.2583,E2 284.3707} C_DIS
LIN {X -126.823,Y 34.2441,Z 152,A 161.432,B 22.3905,C -1.0424,E1 22.2594,E2 285.9203} C_DIS
LIN {X -125.9039,Y 37.4849,Z 152,A 160.1372,B 22.39,C -1.0542,E1 22.2604,E2 287.1923} C_DIS
LIN {X -124.6731,Y 41.3904,Z 152,A 158.492,B 22.3895,C -1.0657,E1 22.2618,E2 288.8178} C_DIS
LIN {X -123.5516,Y 44.6267,Z 152,A 156.7064,B 22.3898,C -1.0581,E1 22.2635,E2 290.6349} C_DIS
LIN {X -122.3833,Y 47.7375,Z 152,A 154.827,B 22.3904,C -1.0447,E1 22.2655,E2 292.5616} C_DIS
LIN {X -120.4073,Y 52.5242,Z 152,A 153.09,B 22.3891,C -1.0732,E1 22.2673,E2 294.2343} C_DIS
LIN {X -118.2379,Y 57.243,Z 152,A 150.6973,B 22.3891,C -1.0746,E1 22.2702,E2 296.6379} C_DIS
LIN {X -116.0864,Y 61.4872,Z 152,A 148.8194,B 22.3884,C -1.089,E1 22.2726,E2 298.4893} C_DIS
LIN {X -114.0011,Y 65.2749,Z 152,A 146.8782,B 22.3883,C -1.0921,E1 22.2752,E2 300.4337} C_DIS
LIN {X -111.8622,Y 68.876,Z 152,A 145.1377,B 22.3879,C -1.1009,E1 22.2777,E2 302.1611} C_DIS
LIN {X -109.3496,Y 72.7992,Z 152,A 142.9857,B 22.3879,C -1.1015,E1 22.281,E2 304.3237} C_DIS
LIN {X -106.864,Y 76.4009,Z 152,A 141.0763,B 22.3876,C -1.1067,E1 22.2841,E2 306.23} C_DIS
LIN {X -104.2075,Y 79.9867,Z 152,A 139.0959,B 22.3874,C -1.1105,E1 22.2874,E2 308.2112} C_DIS
LIN {X -101.425,Y 83.4874,Z 152,A 137.1297,B 22.3872,C -1.1149,E1 22.2908,E2 310.1762} C_DIS
LIN {X -98.657,Y 86.7407,Z 152,A 135.2296,B 22.3871,C -1.1181,E1 22.2943,E2 312.0776} C_DIS
LIN {X -95.6051,Y 90.0926,Z 152,A 133.2832,B 22.3868,C -1.1243,E1 22.298,E2 314.0173} C_DIS
LIN {X -92.4619,Y 93.3159,Z 152,A 131.3158,B 22.3865,C -1.1288,E1 22.3019,E2 315.9821} C_DIS
LIN {X -89.2344,Y 96.4074,Z 152,A 129.3154,B 22.3865,C -1.1312,E1 22.3059,E2 317.9855} C_DIS
LIN {X -85.9443,Y 99.3512,Z 152,A 127.3753,B 22.3863,C -1.1349,E1 22.31,E2 319.9245} C_DIS
LIN {X -82.4248,Y 102.2897,Z 152,A 125.4146,B 22.386,C -1.1409,E1 22.3142,E2 321.8777} C_DIS
LIN {X -78.9824,Y 104.9707,Z 152,A 123.4927,B 22.3858,C -1.1441,E1 22.3185,E2 323.7992} C_DIS
LIN {X -75.4301,Y 107.5521,Z 152,A 121.5713,B 22.3856,C -1.1477,E1 22.3228,E2 325.7187} C_DIS
LIN {X -70.8893,Y 110.5972,Z 152,A 119.1754,B 22.3854,C -1.1518,E1 22.3284,E2 328.1127} C_DIS
LIN {X -67.0252,Y 112.9811,Z 152,A 117.1679,B 22.3854,C -1.1542,E1 22.3332,E2 330.1209} C_DIS
LIN {X -63.429,Y 115.0384,Z 152,A 115.3278,B 22.3852,C -1.1559,E1 22.3377,E2 331.9625} C_DIS
LIN {X -60.0943,Y 116.8139,Z 152,A 113.903,B 22.3846,C -1.1682,E1 22.3411,E2 333.3592} C_DIS
LIN {X -56.8768,Y 118.4129,Z 152,A 112.4513,B 22.3843,C -1.1757,E1 22.3447,E2 334.7955} C_DIS
LIN {X -54.6133,Y 119.4748,Z 152,A 110.3792,B 22.3863,C -1.1349,E1 22.3503,E2 336.9807} C_DIS
LIN {X -49.5422,Y 121.6647,Z 152,A 108.6874,B 22.3846,C -1.1692,E1 22.3544,E2 338.5865} C_DIS
LIN {X -46.4999,Y 122.8596,Z 152,A 107.0908,B 22.3849,C -1.1637,E1 22.3586,E2 340.2017} C_DIS
LIN {X -41.8042,Y 124.5353,Z 152,A 105.0499,B 22.3844,C -1.1721,E1 22.364,E2 342.2247} C_DIS
LIN {X -38.724,Y 125.5272,Z 152,A 103.7993,B 22.384,C -1.1808,E1 22.3673,E2 343.4551} C_DIS
LIN {X -35.6023,Y 126.448,Z 152,A 102.2255,B 22.3843,C -1.1755,E1 22.3715,E2 345.0456} C_DIS
LIN {X -32.0908,Y 127.3845,Z 152,A 100.6091,B 22.3843,C -1.1757,E1 22.3759,E2 346.6643} C_DIS
LIN {X -29.3214,Y 128.0501,Z 152,A 98.9739,B 22.3851,C -1.1595,E1 22.3805,E2 348.3443} C_DIS
LIN {X -25.2763,Y 128.9111,Z 152,A 97.6501,B 22.3839,C -1.182,E1 22.3839,E2 349.6106} C_DIS
LIN {X -21.7159,Y 129.557,Z 152,A 96.0435,B 22.3839,C -1.182,E1 22.3884,E2 351.2192} C_DIS
LIN {X -18.3338,Y 130.079,Z 152,A 94.5232,B 22.3839,C -1.1817,E1 22.3926,E2 352.7417} C_DIS
LIN {X -14.1216,Y 130.6032,Z 152,A 92.4047,B 22.3845,C -1.1708,E1 22.3985,E2 354.8903} C_DIS
LIN {X -8.4702,Y 131.0918,Z 152,A 90.1896,B 22.3839,C -1.1834,E1 22.4046,E2 357.0734} C_DIS
LIN {X -4.9293,Y 131.2722,Z 152,A 88.6118,B 22.3839,C -1.1825,E1 22.409,E2 358.654} C_DIS
LIN {X -1.2253,Y 131.3599,Z 152,A 86.9219,B 22.3841,C -1.1795,E1 22.4138,E2 360.3518} C_DIS
LIN {X 3.3362,Y 131.3226,Z 152,A 84.8861,B 22.3841,C -1.1777,E1 22.4195,E2 362.3921} C_DIS
LIN {X 8.0403,Y 131.1182,Z 152,A 82.9874,B 22.3838,C -1.1846,E1 22.4247,E2 364.2717} C_DIS
LIN {X 12.0769,Y 130.809,Z 152,A 81.1855,B 22.3839,C -1.1828,E1 22.4297,E2 366.0772} C_DIS
LIN {X 15.571,Y 130.4383,Z 152,A 79.7654,B 22.3837,C -1.1876,E1 22.4336,E2 367.4836} C_DIS
LIN {X 19.5502,Y 129.9027,Z 152,A 77.9063,B 22.3839,C -1.1822,E1 22.4388,E2 369.355} C_DIS
LIN {X 22.8671,Y 129.3591,Z 152,A 76.5022,B 22.3839,C -1.1845,E1 22.4426,E2 370.7515} C_DIS
LIN {X 27.1742,Y 128.5241,Z 152,A 74.0572,B 22.3851,C -1.1595,E1 22.4495,E2 373.2587} C_DIS
LIN {X 31.5347,Y 127.5254,Z 152,A 72.5068,B 22.3842,C -1.1765,E1 22.4536,E2 374.7619} C_DIS
LIN {X 35.2603,Y 126.5436,Z 152,A 70.9142,B 22.3841,C -1.1794,E1 22.4578,E2 376.344} C_DIS
Enddeposition()
END
